SPLINE
SPL {X  -165.650, Y  +580.077, Z    +0.000, E1   -64.018, E3 +192650.768}
SPL {X  -165.650, Y  +590.532, Z    +0.000, E1   -63.993, E3 +192661.334}
SPL {X  -165.650, Y  +600.616, Z    +0.000, E1   -64.059, E3 +192670.908}
SPL {X  -165.650, Y  +609.299, Z    +0.000, E1   -64.001, E3 +192679.933}
SPL {X  -165.650, Y  +618.778, Z    +0.000, E1   -63.957, E3 +192689.790}
SPL {X  -165.650, Y  +634.916, Z    +0.000, E1   -64.117, E3 +192704.838}
SPL {X  -165.650, Y  +648.710, Z    +0.000, E1   -63.999, E3 +192719.249}
SPL {X  -165.650, Y  +658.618, Z    +0.000, E1   -64.006, E3 +192729.066}
SPL {X  -165.650, Y  +670.604, Z    +0.000, E1   -64.021, E3 +192740.979}
SPL {X  -165.270, Y  +686.708, Z    +0.000, E1   -64.001, E3 +192757.322}
SPL {X  -163.641, Y  +701.218, Z    +0.000, E1   -63.638, E3 +192774.466}
SPL {X  -161.003, Y  +714.463, Z    +0.000, E1   -63.428, E3 +192789.138}
SPL {X  -157.854, Y  +725.721, Z    +0.000, E1   -62.989, E3 +192803.387}
SPL {X  -155.984, Y  +731.258, Z    +0.000, E1   -62.241, E3 +192813.532}
SPL {X  -153.281, Y  +738.308, Z    +0.000, E1   -62.233, E3 +192820.720}
SPL {X  -150.070, Y  +745.636, Z    +0.000, E1   -61.982, E3 +192829.467}
SPL {X  -146.912, Y  +752.029, Z    +0.000, E1   -61.155, E3 +192840.569}
SPL {X  -143.078, Y  +758.979, Z    +0.000, E1   -60.553, E3 +192850.549}
SPL {X  -139.815, Y  +764.336, Z    +0.000, E1   -60.025, E3 +192858.400}
SPL {X  -130.672, Y  +777.307, Z    +0.000, E1   -63.098, E3 +192856.691}
SPL {X   -84.123, Y  +818.200, Z    +0.000, E1   -55.499, E3 +192970.205}
ENDSPLINE

SPLINE
SPL {X  -116.242, Y  +793.515, Z    +0.000, E1   -51.439, E3 +193088.077}
SPL {X  -136.975, Y  +768.655, Z    +0.000, E1   -47.464, E3 +193112.533}
SPL {X  -151.617, Y  +742.224, Z    +0.000, E1   -39.442, E3 +193118.920}
SPL {X  -159.277, Y  +721.007, Z    +0.000, E1   -30.118, E3 +193118.098}
SPL {X  -163.701, Y  +700.836, Z    +0.000, E1   -18.960, E3 +193114.812}
SPL {X  -165.229, Y  +687.300, Z    +0.000, E1   -10.302, E3 +193114.768}
SPL {X  -165.635, Y  +677.721, Z    +0.000, E1    -3.517, E3 +193113.899}
SPL {X  -165.650, Y  +672.966, Z    +0.000, E1    +0.394, E3 +193112.802}
SPL {X  -165.650, Y  +668.094, Z    +0.000, E1    +7.098, E3 +193111.985}
SPL {X  -165.650, Y  +662.291, Z    +0.000, E1   +16.729, E3 +193111.910}
SPL {X  -165.650, Y  +656.382, Z    +0.000, E1   +26.732, E3 +193111.468}
SPL {X  -165.650, Y  +648.240, Z    +0.000, E1   +42.276, E3 +193106.902}
SPL {X  -165.650, Y  +638.477, Z    +0.000, E1   +48.488, E3 +193113.403}
SPL {X  -165.650, Y  +615.287, Z    +0.000, E1   +74.123, E3 +193097.934}
SPL {X  -165.650, Y  +589.967, Z    +0.000, E1   +71.395, E3 +193114.277}
SPL {X  -165.650, Y  +573.012, Z    +0.000, E1   +68.475, E3 +193130.490}
SPL {X  -165.650, Y  +459.505, Z    +0.000, E1   +68.780, E3 +193202.214}
ENDSPLINE

SPLINE
SPL {X  -165.650, Y  +483.715, Z    +0.000, E1   +63.891, E3 +193218.508}
ENDSPLINE

SPLINE
SPL {X  -165.650, Y  +474.626, Z    +0.000, E1   +63.707, E3 +193229.037}
SPL {X  -165.650, Y  +465.190, Z    +0.000, E1   +63.660, E3 +193238.892}
SPL {X  -165.650, Y  +456.011, Z    +0.000, E1   +63.585, E3 +193248.786}
SPL {X  -165.650, Y  +444.310, Z    +0.000, E1   +63.666, E3 +193260.064}
SPL {X  -165.650, Y  +429.845, Z    +0.000, E1   +64.481, E3 +193268.297}
SPL {X  -165.552, Y  +372.799, Z    +0.000, E1   +69.633, E3 +193274.161}
SPL {X  -165.443, Y  +370.231, Z    +0.000, E1   +68.724, E3 +193284.091}
SPL {X  -164.908, Y  +362.840, Z    +0.000, E1   +68.443, E3 +193292.436}
SPL {X  -164.361, Y  +357.877, Z    +0.000, E1   +67.700, E3 +193302.891}
SPL {X  -163.803, Y  +353.836, Z    +0.000, E1   +66.282, E3 +193317.912}
SPL {X  -163.046, Y  +349.241, Z    +0.000, E1   +65.245, E3 +193329.838}
SPL {X  -160.229, Y  +336.468, Z    +0.000, E1   +65.236, E3 +193341.821}
SPL {X  -157.078, Y  +325.903, Z    +0.000, E1   +64.692, E3 +193355.266}
SPL {X  -154.296, Y  +318.230, Z    +0.000, E1   +64.302, E3 +193364.823}
SPL {X  -151.091, Y  +310.592, Z    +0.000, E1   +63.929, E3 +193374.274}
SPL {X  -148.836, Y  +305.783, Z    +0.000, E1   +63.120, E3 +193383.406}
SPL {X  -145.492, Y  +299.305, Z    +0.000, E1   +63.037, E3 +193389.898}
SPL {X  -142.120, Y  +293.401, Z    +0.000, E1   +62.602, E3 +193397.578}
SPL {X  -139.854, Y  +289.726, Z    +0.000, E1   +61.679, E3 +193405.483}
SPL {X  -135.997, Y  +283.923, Z    +0.000, E1   +62.034, E3 +193409.132}
SPL {X  -124.991, Y  +269.793, Z    +0.000, E1   +65.852, E3 +193404.122}
SPL {X   -80.641, Y  +233.804, Z    +0.000, E1   +55.283, E3 +193535.236}
ENDSPLINE

SPLINE
SPL {X  -132.197, Y  +278.681, Z    +0.000, E1   +49.692, E3 +193669.109}
SPL {X  -156.075, Y  +322.998, Z    +0.000, E1   +35.140, E3 +193674.190}
SPL {X  -162.799, Y  +347.901, Z    +0.000, E1   +22.644, E3 +193676.696}
SPL {X  -164.930, Y  +363.071, Z    +0.000, E1   +13.041, E3 +193674.436}
SPL {X  -165.571, Y  +373.394, Z    +0.000, E1    +5.725, E3 +193674.777}
SPL {X  -165.650, Y  +380.325, Z    +0.000, E1    +0.301, E3 +193673.073}
SPL {X  -165.650, Y  +383.460, Z    +0.000, E1    -3.790, E3 +193672.300}
SPL {X  -165.650, Y  +389.311, Z    +0.000, E1   -13.234, E3 +193671.785}
SPL {X  -165.650, Y  +395.103, Z    +0.000, E1   -23.932, E3 +193671.078}
SPL {X  -165.650, Y  +401.925, Z    +0.000, E1   -35.470, E3 +193670.345}
SPL {X  -165.650, Y  +410.900, Z    +0.000, E1   -46.977, E3 +193670.962}
SPL {X  -165.650, Y  +423.066, Z    +0.000, E1   -61.140, E3 +193666.693}
SPL {X  -165.650, Y  +461.121, Z    +0.000, E1   -74.504, E3 +193668.042}
SPL {X  -165.650, Y  +487.674, Z    +0.000, E1   -70.215, E3 +193690.853}
SPL {X  -165.650, Y  +585.482, Z    +0.000, E1   -67.026, E3 +193770.016}
ENDSPLINE

SPLINE
SPL {X  -165.650, Y  +571.836, Z    +0.000, E1   -64.066, E3 +193780.036}
ENDSPLINE

SPLINE
SPL {X  -165.650, Y  +580.077, Z    +0.000, E1   -64.018, E3 +193788.699}
SPL {X  -165.650, Y  +590.532, Z    +0.000, E1   -63.993, E3 +193799.265}
SPL {X  -165.650, Y  +604.471, Z    +0.000, E1   -64.071, E3 +193812.773}
SPL {X  -165.650, Y  +618.778, Z    +0.000, E1   -63.957, E3 +193827.721}
SPL {X  -165.650, Y  +627.902, Z    +0.000, E1   -63.871, E3 +193837.447}
SPL {X  -165.650, Y  +640.120, Z    +0.000, E1   -64.248, E3 +193846.788}
SPL {X  -165.650, Y  +648.710, Z    +0.000, E1   -63.999, E3 +193857.180}
SPL {X  -165.650, Y  +660.990, Z    +0.000, E1   -63.976, E3 +193869.705}
SPL {X  -165.633, Y  +677.852, Z    +0.000, E1   -63.999, E3 +193886.478}
SPL {X  -164.651, Y  +693.668, Z    +0.000, E1   -63.860, E3 +193903.310}
SPL {X  -162.406, Y  +708.122, Z    +0.000, E1   -63.726, E3 +193918.604}
SPL {X  -159.930, Y  +718.656, Z    +0.000, E1   -63.142, E3 +193933.215}
SPL {X  -156.651, Y  +729.355, Z    +0.000, E1   -62.675, E3 +193947.051}
SPL {X  -153.281, Y  +738.308, Z    +0.000, E1   -62.233, E3 +193958.651}
SPL {X  -150.070, Y  +745.636, Z    +0.000, E1   -61.982, E3 +193967.398}
SPL {X  -146.912, Y  +752.029, Z    +0.000, E1   -61.155, E3 +193978.500}
SPL {X  -143.078, Y  +758.979, Z    +0.000, E1   -60.553, E3 +193988.480}
SPL {X  -139.815, Y  +764.336, Z    +0.000, E1   -60.025, E3 +193996.332}
SPL {X  -133.503, Y  +773.566, Z    +0.000, E1   -62.412, E3 +193994.458}
SPL {X  -122.896, Y  +786.569, Z    +0.000, E1   -64.831, E3 +193994.618}
SPL {X   -84.123, Y  +818.200, Z    +0.000, E1   -55.499, E3 +194108.136}
ENDSPLINE

SPLINE
SPL {X  -127.502, Y  +781.251, Z    +0.000, E1   -49.821, E3 +194240.269}
SPL {X  -156.175, Y  +730.721, Z    +0.000, E1   -34.737, E3 +194256.548}
SPL {X  -163.040, Y  +704.788, Z    +0.000, E1   -21.201, E3 +194252.248}
SPL {X  -165.038, Y  +689.727, Z    +0.000, E1   -11.987, E3 +194252.895}
SPL {X  -165.635, Y  +677.721, Z    +0.000, E1    -3.517, E3 +194251.830}
SPL {X  -165.650, Y  +672.966, Z    +0.000, E1    +0.394, E3 +194250.733}
SPL {X  -165.650, Y  +668.094, Z    +0.000, E1    +7.098, E3 +194249.916}
SPL {X  -165.650, Y  +661.377, Z    +0.000, E1   +18.170, E3 +194249.856}
SPL {X  -165.650, Y  +654.692, Z    +0.000, E1   +29.740, E3 +194249.104}
SPL {X  -165.650, Y  +648.240, Z    +0.000, E1   +42.276, E3 +194244.833}
SPL {X  -165.650, Y  +638.477, Z    +0.000, E1   +48.488, E3 +194251.334}
SPL {X  -165.650, Y  +615.287, Z    +0.000, E1   +74.123, E3 +194235.865}
SPL {X  -165.650, Y  +589.967, Z    +0.000, E1   +71.395, E3 +194252.208}
SPL {X  -165.650, Y  +573.012, Z    +0.000, E1   +68.475, E3 +194268.421}
SPL {X  -165.650, Y  +459.505, Z    +0.000, E1   +68.780, E3 +194340.145}
ENDSPLINE

SPLINE
SPL {X  -165.650, Y  +483.715, Z    +0.000, E1   +63.891, E3 +194356.439}
ENDSPLINE

SPLINE
SPL {X  -165.650, Y  +474.626, Z    +0.000, E1   +63.707, E3 +194366.968}
SPL {X  -165.650, Y  +465.190, Z    +0.000, E1   +63.660, E3 +194376.823}
SPL {X  -165.650, Y  +456.011, Z    +0.000, E1   +63.585, E3 +194386.717}
SPL {X  -165.650, Y  +441.325, Z    +0.000, E1   +63.847, E3 +194399.687}
SPL {X  -165.552, Y  +372.799, Z    +0.000, E1   +69.633, E3 +194412.092}
SPL {X  -165.443, Y  +370.231, Z    +0.000, E1   +68.724, E3 +194422.022}
SPL {X  -164.776, Y  +361.504, Z    +0.000, E1   +68.225, E3 +194433.497}
SPL {X  -164.241, Y  +356.944, Z    +0.000, E1   +66.930, E3 +194448.020}
SPL {X  -163.312, Y  +350.765, Z    +0.000, E1   +66.182, E3 +194459.196}
SPL {X  -163.046, Y  +349.241, Z    +0.000, E1   +65.245, E3 +194467.769}
SPL {X  -160.229, Y  +336.468, Z    +0.000, E1   +65.236, E3 +194479.752}
SPL {X  -157.078, Y  +325.903, Z    +0.000, E1   +64.692, E3 +194493.197}
SPL {X  -153.279, Y  +315.688, Z    +0.000, E1   +64.219, E3 +194505.770}
SPL {X  -149.447, Y  +307.046, Z    +0.000, E1   +63.460, E3 +194518.355}
SPL {X  -145.492, Y  +299.305, Z    +0.000, E1   +63.037, E3 +194527.829}
SPL {X  -142.120, Y  +293.401, Z    +0.000, E1   +62.602, E3 +194535.509}
SPL {X  -139.854, Y  +289.726, Z    +0.000, E1   +61.679, E3 +194543.414}
SPL {X  -135.997, Y  +283.923, Z    +0.000, E1   +62.034, E3 +194547.064}
SPL {X  -124.991, Y  +269.793, Z    +0.000, E1   +65.852, E3 +194542.053}
SPL {X   -80.641, Y  +233.804, Z    +0.000, E1   +55.283, E3 +194673.167}
ENDSPLINE

SPLINE
SPL {X  -132.197, Y  +278.681, Z    +0.000, E1   +49.692, E3 +194807.040}
SPL {X  -156.075, Y  +322.998, Z    +0.000, E1   +35.140, E3 +194812.121}
SPL {X  -162.799, Y  +347.901, Z    +0.000, E1   +22.644, E3 +194814.627}
SPL {X  -164.930, Y  +363.071, Z    +0.000, E1   +13.041, E3 +194812.367}
SPL {X  -165.629, Y  +375.893, Z    +0.000, E1    +3.908, E3 +194812.224}
SPL {X  -165.650, Y  +380.596, Z    +0.000, E1    -0.052, E3 +194810.906}
SPL {X  -165.650, Y  +383.460, Z    +0.000, E1    -3.790, E3 +194810.231}
SPL {X  -165.650, Y  +389.311, Z    +0.000, E1   -13.234, E3 +194809.716}
SPL {X  -165.650, Y  +395.103, Z    +0.000, E1   -23.932, E3 +194809.009}
SPL {X  -165.650, Y  +401.925, Z    +0.000, E1   -35.470, E3 +194808.276}
SPL {X  -165.650, Y  +410.900, Z    +0.000, E1   -46.977, E3 +194808.893}
SPL {X  -165.650, Y  +420.865, Z    +0.000, E1   -58.704, E3 +194805.785}
SPL {X  -165.650, Y  +450.181, Z    +0.000, E1   -73.218, E3 +194803.732}
SPL {X  -165.650, Y  +487.674, Z    +0.000, E1   -70.215, E3 +194828.784}
SPL {X  -165.650, Y  +590.449, Z    +0.000, E1   -68.990, E3 +194896.729}
ENDSPLINE

SPLINE
SPL {X  -165.650, Y  +577.071, Z    +0.000, E1   -65.152, E3 +194915.052}
ENDSPLINE

SPLINE
SPL {X  -165.650, Y  +580.077, Z    +0.000, E1   -64.018, E3 +194926.630}
SPL {X  -165.650, Y  +590.532, Z    +0.000, E1   -63.993, E3 +194937.196}
SPL {X  -165.650, Y  +600.616, Z    +0.000, E1   -64.059, E3 +194946.770}
SPL {X  -165.650, Y  +609.299, Z    +0.000, E1   -64.001, E3 +194955.795}
SPL {X  -165.650, Y  +618.778, Z    +0.000, E1   -63.957, E3 +194965.652}
SPL {X  -165.650, Y  +634.916, Z    +0.000, E1   -64.117, E3 +194980.700}
SPL {X  -165.650, Y  +648.710, Z    +0.000, E1   -63.999, E3 +194995.111}
SPL {X  -165.650, Y  +658.618, Z    +0.000, E1   -64.006, E3 +195004.928}
SPL {X  -165.650, Y  +670.604, Z    +0.000, E1   -64.021, E3 +195016.841}
SPL {X  -165.270, Y  +686.708, Z    +0.000, E1   -64.001, E3 +195033.184}
SPL {X  -163.641, Y  +701.218, Z    +0.000, E1   -63.638, E3 +195050.328}
SPL {X  -161.003, Y  +714.463, Z    +0.000, E1   -63.428, E3 +195065.000}
SPL {X  -157.854, Y  +725.721, Z    +0.000, E1   -62.989, E3 +195079.249}
SPL {X  -155.984, Y  +731.258, Z    +0.000, E1   -62.241, E3 +195089.395}
SPL {X  -153.281, Y  +738.308, Z    +0.000, E1   -62.233, E3 +195096.582}
SPL {X  -150.070, Y  +745.636, Z    +0.000, E1   -61.982, E3 +195105.329}
SPL {X  -148.438, Y  +749.026, Z    +0.000, E1   -61.150, E3 +195113.335}
SPL {X  -145.760, Y  +754.202, Z    +0.000, E1   -61.108, E3 +195118.752}
SPL {X  -143.078, Y  +758.979, Z    +0.000, E1   -60.553, E3 +195126.411}
SPL {X  -139.815, Y  +764.336, Z    +0.000, E1   -60.025, E3 +195134.263}
SPL {X  -130.672, Y  +777.307, Z    +0.000, E1   -63.098, E3 +195132.553}
SPL {X   -84.123, Y  +818.200, Z    +0.000, E1   -55.499, E3 +195246.067}
ENDSPLINE

SPLINE
SPL {X  -127.502, Y  +781.251, Z    +0.000, E1   -49.821, E3 +195378.200}
SPL {X  -151.617, Y  +742.224, Z    +0.000, E1   -39.442, E3 +195394.782}
SPL {X  -159.277, Y  +721.007, Z    +0.000, E1   -30.118, E3 +195393.960}
SPL {X  -163.701, Y  +700.836, Z    +0.000, E1   -18.960, E3 +195390.674}
SPL {X  -165.229, Y  +687.300, Z    +0.000, E1   -10.302, E3 +195390.630}
SPL {X  -165.592, Y  +679.896, Z    +0.000, E1    -5.071, E3 +195389.910}
SPL {X  -165.650, Y  +674.350, Z    +0.000, E1    -0.828, E3 +195389.284}
SPL {X  -165.650, Y  +672.653, Z    +0.000, E1    +0.827, E3 +195388.477}
SPL {X  -165.650, Y  +668.094, Z    +0.000, E1    +7.098, E3 +195387.847}
SPL {X  -165.650, Y  +662.291, Z    +0.000, E1   +16.729, E3 +195387.772}
SPL {X  -165.650, Y  +656.382, Z    +0.000, E1   +26.732, E3 +195387.330}
SPL {X  -165.650, Y  +648.240, Z    +0.000, E1   +42.276, E3 +195382.765}
SPL {X  -165.650, Y  +638.782, Z    +0.000, E1   +47.719, E3 +195389.974}
SPL {X  -165.650, Y  +622.329, Z    +0.000, E1   +68.753, E3 +195377.514}
SPL {X  -165.650, Y  +589.967, Z    +0.000, E1   +71.395, E3 +195390.139}
SPL {X  -165.650, Y  +573.012, Z    +0.000, E1   +68.475, E3 +195406.352}
SPL {X  -165.650, Y  +459.505, Z    +0.000, E1   +68.780, E3 +195478.076}
ENDSPLINE

SPLINE
SPL {X  -165.650, Y  +483.715, Z    +0.000, E1   +63.891, E3 +195494.370}
ENDSPLINE

SPLINE
SPL {X  -165.650, Y  +474.626, Z    +0.000, E1   +63.707, E3 +195504.899}
SPL {X  -165.650, Y  +465.190, Z    +0.000, E1   +63.660, E3 +195514.754}
SPL {X  -165.650, Y  +456.011, Z    +0.000, E1   +63.585, E3 +195524.648}
SPL {X  -165.650, Y  +444.310, Z    +0.000, E1   +63.666, E3 +195535.926}
SPL {X  -165.650, Y  +429.845, Z    +0.000, E1   +64.481, E3 +195544.159}
SPL {X  -165.552, Y  +372.799, Z    +0.000, E1   +69.633, E3 +195550.023}
SPL {X  -165.188, Y  +366.130, Z    +0.000, E1   +68.611, E3 +195564.426}
SPL {X  -164.361, Y  +357.877, Z    +0.000, E1   +67.700, E3 +195578.753}
SPL {X  -163.803, Y  +353.836, Z    +0.000, E1   +66.282, E3 +195593.774}
SPL {X  -162.254, Y  +345.129, Z    +0.000, E1   +65.301, E3 +195609.224}
SPL {X  -158.875, Y  +331.610, Z    +0.000, E1   +64.945, E3 +195624.283}
SPL {X  -154.872, Y  +319.724, Z    +0.000, E1   +64.496, E3 +195638.197}
SPL {X  -151.091, Y  +310.592, Z    +0.000, E1   +63.929, E3 +195650.136}
SPL {X  -148.836, Y  +305.783, Z    +0.000, E1   +63.120, E3 +195659.268}
SPL {X  -145.492, Y  +299.305, Z    +0.000, E1   +63.037, E3 +195665.760}
SPL {X  -142.120, Y  +293.401, Z    +0.000, E1   +62.602, E3 +195673.440}
SPL {X  -139.854, Y  +289.726, Z    +0.000, E1   +61.679, E3 +195681.345}
SPL {X  -135.997, Y  +283.923, Z    +0.000, E1   +62.034, E3 +195684.995}
SPL {X  -124.991, Y  +269.793, Z    +0.000, E1   +65.852, E3 +195679.984}
SPL {X   -80.641, Y  +233.804, Z    +0.000, E1   +55.283, E3 +195811.098}
ENDSPLINE

SPLINE
SPL {X  -132.197, Y  +278.681, Z    +0.000, E1   +49.692, E3 +195944.971}
SPL {X  -156.075, Y  +322.998, Z    +0.000, E1   +35.140, E3 +195950.052}
SPL {X  -162.799, Y  +347.901, Z    +0.000, E1   +22.644, E3 +195952.558}
SPL {X  -164.930, Y  +363.071, Z    +0.000, E1   +13.041, E3 +195950.298}
SPL {X  -165.629, Y  +375.893, Z    +0.000, E1    +3.908, E3 +195950.155}
SPL {X  -165.650, Y  +380.596, Z    +0.000, E1    -0.052, E3 +195948.837}
SPL {X  -165.650, Y  +383.460, Z    +0.000, E1    -3.790, E3 +195948.162}
SPL {X  -165.650, Y  +389.311, Z    +0.000, E1   -13.234, E3 +195947.647}
SPL {X  -165.650, Y  +395.103, Z    +0.000, E1   -23.932, E3 +195946.940}
SPL {X  -165.650, Y  +401.925, Z    +0.000, E1   -35.470, E3 +195946.207}
SPL {X  -165.650, Y  +410.900, Z    +0.000, E1   -46.977, E3 +195946.824}
SPL {X  -165.650, Y  +423.066, Z    +0.000, E1   -61.140, E3 +195942.555}
SPL {X  -165.650, Y  +461.121, Z    +0.000, E1   -74.504, E3 +195943.904}
SPL {X  -165.650, Y  +487.674, Z    +0.000, E1   -70.215, E3 +195966.715}
SPL {X  -165.650, Y  +585.482, Z    +0.000, E1   -67.026, E3 +196045.878}
ENDSPLINE

SPLINE
SPL {X  -165.650, Y  +571.836, Z    +0.000, E1   -64.066, E3 +196055.898}
ENDSPLINE

SPLINE
SPL {X  -165.650, Y  +580.077, Z    +0.000, E1   -64.018, E3 +196064.561}
SPL {X  -165.650, Y  +590.532, Z    +0.000, E1   -63.993, E3 +196075.127}
SPL {X  -165.650, Y  +604.471, Z    +0.000, E1   -64.071, E3 +196088.635}
SPL {X  -165.650, Y  +618.778, Z    +0.000, E1   -63.957, E3 +196103.583}
SPL {X  -165.650, Y  +627.902, Z    +0.000, E1   -63.871, E3 +196113.309}
SPL {X  -165.650, Y  +640.120, Z    +0.000, E1   -64.248, E3 +196122.650}
SPL {X  -165.650, Y  +648.710, Z    +0.000, E1   -63.999, E3 +196133.042}
SPL {X  -165.650, Y  +660.990, Z    +0.000, E1   -63.976, E3 +196145.567}
SPL {X  -165.633, Y  +677.852, Z    +0.000, E1   -63.999, E3 +196162.340}
SPL {X  -164.651, Y  +693.668, Z    +0.000, E1   -63.860, E3 +196179.173}
SPL {X  -162.406, Y  +708.122, Z    +0.000, E1   -63.726, E3 +196194.467}
SPL {X  -159.930, Y  +718.656, Z    +0.000, E1   -63.142, E3 +196209.077}
SPL {X  -156.651, Y  +729.355, Z    +0.000, E1   -62.675, E3 +196222.913}
SPL {X  -153.281, Y  +738.308, Z    +0.000, E1   -62.233, E3 +196234.513}
SPL {X  -150.070, Y  +745.636, Z    +0.000, E1   -61.982, E3 +196243.260}
SPL {X  -148.438, Y  +749.026, Z    +0.000, E1   -61.150, E3 +196251.266}
SPL {X  -145.760, Y  +754.202, Z    +0.000, E1   -61.108, E3 +196256.683}
SPL {X  -143.078, Y  +758.979, Z    +0.000, E1   -60.553, E3 +196264.342}
SPL {X  -139.815, Y  +764.336, Z    +0.000, E1   -60.025, E3 +196272.194}
SPL {X  -130.672, Y  +777.307, Z    +0.000, E1   -63.098, E3 +196270.484}
SPL {X   -84.123, Y  +818.200, Z    +0.000, E1   -55.499, E3 +196383.998}
ENDSPLINE

SPLINE
SPL {X  -116.242, Y  +793.515, Z    +0.000, E1   -51.439, E3 +196501.871}
SPL {X  -136.975, Y  +768.655, Z    +0.000, E1   -47.464, E3 +196526.326}
SPL {X  -151.617, Y  +742.224, Z    +0.000, E1   -39.442, E3 +196532.713}
SPL {X  -159.277, Y  +721.007, Z    +0.000, E1   -30.118, E3 +196531.891}
SPL {X  -163.701, Y  +700.836, Z    +0.000, E1   -18.960, E3 +196528.605}
SPL {X  -165.229, Y  +687.300, Z    +0.000, E1   -10.302, E3 +196528.561}
SPL {X  -165.635, Y  +677.721, Z    +0.000, E1    -3.517, E3 +196527.692}
SPL {X  -165.650, Y  +673.529, Z    +0.000, E1    -0.069, E3 +196526.820}
SPL {X  -165.650, Y  +671.950, Z    +0.000, E1    +1.795, E3 +196526.189}
SPL {X  -165.650, Y  +668.094, Z    +0.000, E1    +7.098, E3 +196525.778}
SPL {X  -165.650, Y  +661.377, Z    +0.000, E1   +18.170, E3 +196525.718}
SPL {X  -165.650, Y  +654.692, Z    +0.000, E1   +29.740, E3 +196524.966}
SPL {X  -165.650, Y  +648.240, Z    +0.000, E1   +42.276, E3 +196520.696}
SPL {X  -165.650, Y  +638.477, Z    +0.000, E1   +48.488, E3 +196527.196}
SPL {X  -165.650, Y  +615.287, Z    +0.000, E1   +74.123, E3 +196511.727}
SPL {X  -165.650, Y  +589.967, Z    +0.000, E1   +71.395, E3 +196528.070}
SPL {X  -165.650, Y  +573.012, Z    +0.000, E1   +68.475, E3 +196544.283}
SPL {X  -165.650, Y  +459.505, Z    +0.000, E1   +68.780, E3 +196616.007}
ENDSPLINE

SPLINE
SPL {X  -165.650, Y  +483.715, Z    +0.000, E1   +63.891, E3 +196632.301}
ENDSPLINE

SPLINE
SPL {X  -165.650, Y  +474.626, Z    +0.000, E1   +63.707, E3 +196642.830}
SPL {X  -165.650, Y  +465.190, Z    +0.000, E1   +63.660, E3 +196652.685}
SPL {X  -165.650, Y  +456.011, Z    +0.000, E1   +63.585, E3 +196662.579}
SPL {X  -165.650, Y  +441.325, Z    +0.000, E1   +63.847, E3 +196675.549}
SPL {X  -165.552, Y  +372.799, Z    +0.000, E1   +69.633, E3 +196687.954}
SPL {X  -165.443, Y  +370.231, Z    +0.000, E1   +68.724, E3 +196697.884}
SPL {X  -164.908, Y  +362.840, Z    +0.000, E1   +68.443, E3 +196706.229}
SPL {X  -164.361, Y  +357.877, Z    +0.000, E1   +67.700, E3 +196716.684}
SPL {X  -163.803, Y  +353.836, Z    +0.000, E1   +66.282, E3 +196731.705}
SPL {X  -162.254, Y  +345.129, Z    +0.000, E1   +65.301, E3 +196747.155}
SPL {X  -158.875, Y  +331.610, Z    +0.000, E1   +64.945, E3 +196762.214}
SPL {X  -154.872, Y  +319.724, Z    +0.000, E1   +64.496, E3 +196776.128}
SPL {X  -151.091, Y  +310.592, Z    +0.000, E1   +63.929, E3 +196788.067}
SPL {X  -148.836, Y  +305.783, Z    +0.000, E1   +63.120, E3 +196797.199}
SPL {X  -145.492, Y  +299.305, Z    +0.000, E1   +63.037, E3 +196803.691}
SPL {X  -142.120, Y  +293.401, Z    +0.000, E1   +62.602, E3 +196811.371}
SPL {X  -139.854, Y  +289.726, Z    +0.000, E1   +61.679, E3 +196819.276}
SPL {X  -135.997, Y  +283.923, Z    +0.000, E1   +62.034, E3 +196822.926}
SPL {X  -124.991, Y  +269.793, Z    +0.000, E1   +65.852, E3 +196817.915}
SPL {X   -80.641, Y  +233.804, Z    +0.000, E1   +55.283, E3 +196949.029}
ENDSPLINE

SPLINE
SPL {X  -126.633, Y  +271.710, Z    +0.000, E1   +51.055, E3 +197079.495}
SPL {X  -147.744, Y  +303.590, Z    +0.000, E1   +42.717, E3 +197087.987}
SPL {X  -158.730, Y  +331.121, Z    +0.000, E1   +31.334, E3 +197087.895}
SPL {X  -162.799, Y  +347.901, Z    +0.000, E1   +22.644, E3 +197090.489}
SPL {X  -164.930, Y  +363.071, Z    +0.000, E1   +13.041, E3 +197088.229}
SPL {X  -165.629, Y  +375.893, Z    +0.000, E1    +3.908, E3 +197088.086}
SPL {X  -165.650, Y  +380.596, Z    +0.000, E1    -0.052, E3 +197086.768}
SPL {X  -165.650, Y  +383.460, Z    +0.000, E1    -3.790, E3 +197086.093}
SPL {X  -165.650, Y  +387.326, Z    +0.000, E1   -10.041, E3 +197085.964}
SPL {X  -165.650, Y  +392.519, Z    +0.000, E1   -19.014, E3 +197085.118}
SPL {X  -165.650, Y  +401.925, Z    +0.000, E1   -35.470, E3 +197084.138}
SPL {X  -165.650, Y  +410.900, Z    +0.000, E1   -46.977, E3 +197084.756}
SPL {X  -165.650, Y  +420.865, Z    +0.000, E1   -58.704, E3 +197081.647}
SPL {X  -165.650, Y  +450.181, Z    +0.000, E1   -73.218, E3 +197079.594}
SPL {X  -165.650, Y  +487.674, Z    +0.000, E1   -70.215, E3 +197104.646}
SPL {X  -165.650, Y  +590.449, Z    +0.000, E1   -68.990, E3 +197172.591}
ENDSPLINE

SPLINE
SPL {X  -165.650, Y  +577.071, Z    +0.000, E1   -65.152, E3 +197190.914}
ENDSPLINE

SPLINE
SPL {X  -165.650, Y  +580.077, Z    +0.000, E1   -64.018, E3 +197202.492}
SPL {X  -165.650, Y  +590.532, Z    +0.000, E1   -63.993, E3 +197213.058}
SPL {X  -165.650, Y  +604.471, Z    +0.000, E1   -64.071, E3 +197226.566}
SPL {X  -165.650, Y  +618.778, Z    +0.000, E1   -63.957, E3 +197241.514}
SPL {X  -165.650, Y  +627.902, Z    +0.000, E1   -63.871, E3 +197251.240}
SPL {X  -165.650, Y  +640.120, Z    +0.000, E1   -64.248, E3 +197260.581}
SPL {X  -165.650, Y  +648.710, Z    +0.000, E1   -63.999, E3 +197270.973}
SPL {X  -165.650, Y  +658.618, Z    +0.000, E1   -64.006, E3 +197280.790}
SPL {X  -165.650, Y  +670.604, Z    +0.000, E1   -64.021, E3 +197292.703}
SPL {X  -165.270, Y  +686.708, Z    +0.000, E1   -64.001, E3 +197309.046}
SPL {X  -164.361, Y  +696.123, Z    +0.000, E1   -63.520, E3 +197321.757}
SPL {X  -162.406, Y  +708.122, Z    +0.000, E1   -63.726, E3 +197332.398}
SPL {X  -159.930, Y  +718.656, Z    +0.000, E1   -63.142, E3 +197347.008}
SPL {X  -157.142, Y  +727.904, Z    +0.000, E1   -62.905, E3 +197357.697}
SPL {X  -154.742, Y  +734.618, Z    +0.000, E1   -62.412, E3 +197367.596}
SPL {X  -150.939, Y  +743.744, Z    +0.000, E1   -61.955, E3 +197379.537}
SPL {X  -146.912, Y  +752.029, Z    +0.000, E1   -61.155, E3 +197392.293}
SPL {X  -143.078, Y  +758.979, Z    +0.000, E1   -60.553, E3 +197402.273}
SPL {X  -139.815, Y  +764.336, Z    +0.000, E1   -60.025, E3 +197410.125}
SPL {X  -130.672, Y  +777.307, Z    +0.000, E1   -63.098, E3 +197408.415}
SPL {X   -84.123, Y  +818.200, Z    +0.000, E1   -55.499, E3 +197521.929}
ENDSPLINE

SPLINE
SPL {X  -127.502, Y  +781.251, Z    +0.000, E1   -49.821, E3 +197654.062}
SPL {X  -156.175, Y  +730.721, Z    +0.000, E1   -34.737, E3 +197670.341}
SPL {X  -163.701, Y  +700.836, Z    +0.000, E1   -18.960, E3 +197666.536}
SPL {X  -165.229, Y  +687.300, Z    +0.000, E1   -10.302, E3 +197666.492}
SPL {X  -165.592, Y  +679.896, Z    +0.000, E1    -5.071, E3 +197665.772}
SPL {X  -165.650, Y  +673.846, Z    +0.000, E1    -0.441, E3 +197664.852}
SPL {X  -165.650, Y  +670.816, Z    +0.000, E1    +3.131, E3 +197664.143}
SPL {X  -165.650, Y  +666.496, Z    +0.000, E1    +9.886, E3 +197663.217}
SPL {X  -165.650, Y  +662.291, Z    +0.000, E1   +16.729, E3 +197663.634}
SPL {X  -165.650, Y  +656.382, Z    +0.000, E1   +26.732, E3 +197663.192}
SPL {X  -165.650, Y  +648.240, Z    +0.000, E1   +42.276, E3 +197658.627}
SPL {X  -165.650, Y  +638.477, Z    +0.000, E1   +48.488, E3 +197665.127}
SPL {X  -165.650, Y  +615.287, Z    +0.000, E1   +74.123, E3 +197649.658}
SPL {X  -165.650, Y  +589.967, Z    +0.000, E1   +71.395, E3 +197666.001}
SPL {X  -165.650, Y  +573.012, Z    +0.000, E1   +68.475, E3 +197682.214}
SPL {X  -165.650, Y  +459.505, Z    +0.000, E1   +68.780, E3 +197753.938}
ENDSPLINE

SPLINE
SPL {X  -165.650, Y  +483.715, Z    +0.000, E1   +63.891, E3 +197770.232}
ENDSPLINE

SPLINE
SPL {X  -165.650, Y  +474.626, Z    +0.000, E1   +63.707, E3 +197780.761}
SPL {X  -165.650, Y  +465.190, Z    +0.000, E1   +63.660, E3 +197790.616}
SPL {X  -165.650, Y  +456.011, Z    +0.000, E1   +63.585, E3 +197800.510}
SPL {X  -165.650, Y  +441.325, Z    +0.000, E1   +63.847, E3 +197813.480}
SPL {X  -165.552, Y  +372.799, Z    +0.000, E1   +69.633, E3 +197825.885}
SPL {X  -165.443, Y  +370.231, Z    +0.000, E1   +68.724, E3 +197835.815}
SPL {X  -164.776, Y  +361.504, Z    +0.000, E1   +68.225, E3 +197847.290}
SPL {X  -164.241, Y  +356.944, Z    +0.000, E1   +66.930, E3 +197861.813}
SPL {X  -163.312, Y  +350.765, Z    +0.000, E1   +66.182, E3 +197872.989}
SPL {X  -163.046, Y  +349.241, Z    +0.000, E1   +65.245, E3 +197881.562}
SPL {X  -160.229, Y  +336.468, Z    +0.000, E1   +65.236, E3 +197893.545}
SPL {X  -157.078, Y  +325.903, Z    +0.000, E1   +64.692, E3 +197906.991}
SPL {X  -153.279, Y  +315.688, Z    +0.000, E1   +64.219, E3 +197919.563}
SPL {X  -149.447, Y  +307.046, Z    +0.000, E1   +63.460, E3 +197932.148}
SPL {X  -145.492, Y  +299.305, Z    +0.000, E1   +63.037, E3 +197941.622}
SPL {X  -142.120, Y  +293.401, Z    +0.000, E1   +62.602, E3 +197949.302}
SPL {X  -139.854, Y  +289.726, Z    +0.000, E1   +61.679, E3 +197957.207}
SPL {X  -135.997, Y  +283.923, Z    +0.000, E1   +62.034, E3 +197960.857}
SPL {X  -124.991, Y  +269.793, Z    +0.000, E1   +65.852, E3 +197955.846}
SPL {X   -80.641, Y  +233.804, Z    +0.000, E1   +55.283, E3 +198086.960}
ENDSPLINE

SPLINE
SPL {X  -126.633, Y  +271.710, Z    +0.000, E1   +51.055, E3 +198217.426}
SPL {X  -147.744, Y  +303.590, Z    +0.000, E1   +42.717, E3 +198225.918}
SPL {X  -158.730, Y  +331.121, Z    +0.000, E1   +31.334, E3 +198225.826}
SPL {X  -162.799, Y  +347.901, Z    +0.000, E1   +22.644, E3 +198228.420}
SPL {X  -164.930, Y  +363.071, Z    +0.000, E1   +13.041, E3 +198226.160}
SPL {X  -165.629, Y  +375.893, Z    +0.000, E1    +3.908, E3 +198226.017}
SPL {X  -165.650, Y  +381.007, Z    +0.000, E1    -0.398, E3 +198224.557}
SPL {X  -165.650, Y  +385.791, Z    +0.000, E1    -7.347, E3 +198223.918}
SPL {X  -165.650, Y  +390.879, Z    +0.000, E1   -16.263, E3 +198223.205}
SPL {X  -165.650, Y  +395.103, Z    +0.000, E1   -23.932, E3 +198222.803}
SPL {X  -165.650, Y  +401.925, Z    +0.000, E1   -35.470, E3 +198222.069}
SPL {X  -165.650, Y  +410.900, Z    +0.000, E1   -46.977, E3 +198222.687}
SPL {X  -165.650, Y  +423.066, Z    +0.000, E1   -61.140, E3 +198218.417}
SPL {X  -165.650, Y  +461.121, Z    +0.000, E1   -74.504, E3 +198219.766}
SPL {X  -165.650, Y  +487.674, Z    +0.000, E1   -70.215, E3 +198242.577}
SPL {X  -165.650, Y  +585.482, Z    +0.000, E1   -67.026, E3 +198321.740}
ENDSPLINE

SPLINE
SPL {X  -165.650, Y  +571.836, Z    +0.000, E1   -64.066, E3 +198331.760}
ENDSPLINE

SPLINE
SPL {X  -165.650, Y  +580.077, Z    +0.000, E1   -64.018, E3 +198340.423}
SPL {X  -165.650, Y  +590.532, Z    +0.000, E1   -63.993, E3 +198350.989}
SPL {X  -165.650, Y  +600.616, Z    +0.000, E1   -64.059, E3 +198360.563}
SPL {X  -165.650, Y  +609.299, Z    +0.000, E1   -64.001, E3 +198369.588}
SPL {X  -165.650, Y  +618.778, Z    +0.000, E1   -63.957, E3 +198379.445}
SPL {X  -165.650, Y  +627.902, Z    +0.000, E1   -63.871, E3 +198389.171}
SPL {X  -165.650, Y  +640.120, Z    +0.000, E1   -64.248, E3 +198398.512}
SPL {X  -165.650, Y  +648.710, Z    +0.000, E1   -63.999, E3 +198408.904}
SPL {X  -165.650, Y  +658.618, Z    +0.000, E1   -64.006, E3 +198418.721}
SPL {X  -165.650, Y  +670.604, Z    +0.000, E1   -64.021, E3 +198430.635}
SPL {X  -165.553, Y  +681.156, Z    +0.000, E1   -63.834, E3 +198442.509}
SPL {X  -164.651, Y  +693.668, Z    +0.000, E1   -63.860, E3 +198455.035}
SPL {X  -163.017, Y  +704.915, Z    +0.000, E1   -63.665, E3 +198467.477}
SPL {X  -161.003, Y  +714.463, Z    +0.000, E1   -63.428, E3 +198478.793}
SPL {X  -157.854, Y  +725.721, Z    +0.000, E1   -62.989, E3 +198493.042}
SPL {X  -155.984, Y  +731.258, Z    +0.000, E1   -62.241, E3 +198503.188}
SPL {X  -153.281, Y  +738.308, Z    +0.000, E1   -62.233, E3 +198510.375}
SPL {X  -150.070, Y  +745.636, Z    +0.000, E1   -61.982, E3 +198519.122}
SPL {X  -146.912, Y  +752.029, Z    +0.000, E1   -61.155, E3 +198530.224}
SPL {X  -143.078, Y  +758.979, Z    +0.000, E1   -60.553, E3 +198540.204}
SPL {X  -139.815, Y  +764.336, Z    +0.000, E1   -60.025, E3 +198548.056}
SPL {X  -130.672, Y  +777.307, Z    +0.000, E1   -63.098, E3 +198546.346}
SPL {X   -84.123, Y  +818.200, Z    +0.000, E1   -55.499, E3 +198659.860}
ENDSPLINE

SPLINE
SPL {X  -127.502, Y  +781.251, Z    +0.000, E1   -49.821, E3 +198791.993}
SPL {X  -151.617, Y  +742.224, Z    +0.000, E1   -39.442, E3 +198808.575}
SPL {X  -159.277, Y  +721.007, Z    +0.000, E1   -30.118, E3 +198807.753}
SPL {X  -163.701, Y  +700.836, Z    +0.000, E1   -18.960, E3 +198804.467}
SPL {X  -165.229, Y  +687.300, Z    +0.000, E1   -10.302, E3 +198804.423}
SPL {X  -165.592, Y  +679.896, Z    +0.000, E1    -5.071, E3 +198803.704}
SPL {X  -165.650, Y  +673.846, Z    +0.000, E1    -0.441, E3 +198802.783}
SPL {X  -165.650, Y  +670.816, Z    +0.000, E1    +3.131, E3 +198802.074}
SPL {X  -165.650, Y  +666.496, Z    +0.000, E1    +9.886, E3 +198801.148}
SPL {X  -165.650, Y  +661.377, Z    +0.000, E1   +18.170, E3 +198801.580}
SPL {X  -165.650, Y  +654.692, Z    +0.000, E1   +29.740, E3 +198800.828}
SPL {X  -165.650, Y  +648.240, Z    +0.000, E1   +42.276, E3 +198796.558}
SPL {X  -165.650, Y  +638.477, Z    +0.000, E1   +48.488, E3 +198803.058}
SPL {X  -165.650, Y  +615.287, Z    +0.000, E1   +74.123, E3 +198787.589}
SPL {X  -165.650, Y  +589.967, Z    +0.000, E1   +71.395, E3 +198803.932}
SPL {X  -165.650, Y  +573.012, Z    +0.000, E1   +68.475, E3 +198820.145}
SPL {X  -165.650, Y  +459.505, Z    +0.000, E1   +68.780, E3 +198891.869}
ENDSPLINE

SPLINE
SPL {X  -165.650, Y  +483.715, Z    +0.000, E1   +63.891, E3 +198908.163}
ENDSPLINE

SPLINE
SPL {X  -165.650, Y  +474.626, Z    +0.000, E1   +63.707, E3 +198918.692}
SPL {X  -165.650, Y  +465.190, Z    +0.000, E1   +63.660, E3 +198928.547}
SPL {X  -165.650, Y  +456.011, Z    +0.000, E1   +63.585, E3 +198938.441}
SPL {X  -165.650, Y  +444.310, Z    +0.000, E1   +63.666, E3 +198949.719}
SPL {X  -165.650, Y  +429.845, Z    +0.000, E1   +64.481, E3 +198957.952}
SPL {X  -165.552, Y  +372.799, Z    +0.000, E1   +69.633, E3 +198963.816}
SPL {X  -165.188, Y  +366.130, Z    +0.000, E1   +68.611, E3 +198978.219}
SPL {X  -164.361, Y  +357.877, Z    +0.000, E1   +67.700, E3 +198992.546}
SPL {X  -163.803, Y  +353.836, Z    +0.000, E1   +66.282, E3 +199007.567}
SPL {X  -162.254, Y  +345.129, Z    +0.000, E1   +65.301, E3 +199023.017}
SPL {X  -159.503, Y  +333.793, Z    +0.000, E1   +65.139, E3 +199034.462}
SPL {X  -157.078, Y  +325.903, Z    +0.000, E1   +64.692, E3 +199044.922}
SPL {X  -153.279, Y  +315.688, Z    +0.000, E1   +64.219, E3 +199057.494}
SPL {X  -149.447, Y  +307.046, Z    +0.000, E1   +63.460, E3 +199070.079}
SPL {X  -145.492, Y  +299.305, Z    +0.000, E1   +63.037, E3 +199079.553}
SPL {X  -142.120, Y  +293.401, Z    +0.000, E1   +62.602, E3 +199087.233}
SPL {X  -139.854, Y  +289.726, Z    +0.000, E1   +61.679, E3 +199095.138}
SPL {X  -135.997, Y  +283.923, Z    +0.000, E1   +62.034, E3 +199098.788}
SPL {X  -124.991, Y  +269.793, Z    +0.000, E1   +65.852, E3 +199093.777}
SPL {X   -80.641, Y  +233.804, Z    +0.000, E1   +55.283, E3 +199224.891}
ENDSPLINE

SPLINE
SPL {X  -132.197, Y  +278.681, Z    +0.000, E1   +49.692, E3 +199358.764}
SPL {X  -156.075, Y  +322.998, Z    +0.000, E1   +35.140, E3 +199363.845}
SPL {X  -163.642, Y  +352.786, Z    +0.000, E1   +19.725, E3 +199365.624}
SPL {X  -165.477, Y  +370.931, Z    +0.000, E1    +7.630, E3 +199364.213}
SPL {X  -165.650, Y  +378.219, Z    +0.000, E1    +1.951, E3 +199363.485}
SPL {X  -165.650, Y  +380.596, Z    +0.000, E1    -0.052, E3 +199362.630}
SPL {X  -165.650, Y  +383.460, Z    +0.000, E1    -3.790, E3 +199361.955}
SPL {X  -165.650, Y  +387.326, Z    +0.000, E1   -10.041, E3 +199361.826}
SPL {X  -165.650, Y  +392.519, Z    +0.000, E1   -19.014, E3 +199360.980}
SPL {X  -165.650, Y  +401.925, Z    +0.000, E1   -35.470, E3 +199360.001}
SPL {X  -165.650, Y  +410.900, Z    +0.000, E1   -46.977, E3 +199360.618}
SPL {X  -165.650, Y  +420.865, Z    +0.000, E1   -58.704, E3 +199357.509}
SPL {X  -165.650, Y  +450.181, Z    +0.000, E1   -73.218, E3 +199355.456}
SPL {X  -165.650, Y  +487.674, Z    +0.000, E1   -70.215, E3 +199380.508}
SPL {X  -165.650, Y  +585.482, Z    +0.000, E1   -67.026, E3 +199459.671}
ENDSPLINE

SPLINE
SPL {X  -165.650, Y  +577.780, Z    +0.000, E1   -64.060, E3 +199475.883}
ENDSPLINE

SPLINE
SPL {X  -165.650, Y  +590.532, Z    +0.000, E1   -63.993, E3 +199488.920}
SPL {X  -165.650, Y  +600.616, Z    +0.000, E1   -64.059, E3 +199498.494}
SPL {X  -165.650, Y  +609.299, Z    +0.000, E1   -64.001, E3 +199507.519}
SPL {X  -165.650, Y  +618.778, Z    +0.000, E1   -63.957, E3 +199517.376}
SPL {X  -165.650, Y  +627.902, Z    +0.000, E1   -63.871, E3 +199527.102}
SPL {X  -165.650, Y  +640.120, Z    +0.000, E1   -64.248, E3 +199536.443}
SPL {X  -165.650, Y  +648.710, Z    +0.000, E1   -63.999, E3 +199546.835}
SPL {X  -165.650, Y  +658.618, Z    +0.000, E1   -64.006, E3 +199556.652}
SPL {X  -165.650, Y  +670.604, Z    +0.000, E1   -64.021, E3 +199568.566}
SPL {X  -165.553, Y  +681.156, Z    +0.000, E1   -63.834, E3 +199580.440}
SPL {X  -164.651, Y  +693.668, Z    +0.000, E1   -63.860, E3 +199592.966}
SPL {X  -163.017, Y  +704.915, Z    +0.000, E1   -63.665, E3 +199605.408}
SPL {X  -161.003, Y  +714.463, Z    +0.000, E1   -63.428, E3 +199616.724}
SPL {X  -157.854, Y  +725.721, Z    +0.000, E1   -62.989, E3 +199630.973}
SPL {X  -155.984, Y  +731.258, Z    +0.000, E1   -62.241, E3 +199641.119}
SPL {X  -153.281, Y  +738.308, Z    +0.000, E1   -62.233, E3 +199648.306}
SPL {X  -150.070, Y  +745.636, Z    +0.000, E1   -61.982, E3 +199657.053}
SPL {X  -148.438, Y  +749.026, Z    +0.000, E1   -61.150, E3 +199665.060}
SPL {X  -145.760, Y  +754.202, Z    +0.000, E1   -61.108, E3 +199670.476}
SPL {X  -143.078, Y  +758.979, Z    +0.000, E1   -60.553, E3 +199678.135}
SPL {X  -139.815, Y  +764.336, Z    +0.000, E1   -60.025, E3 +199685.987}
SPL {X  -130.672, Y  +777.307, Z    +0.000, E1   -63.098, E3 +199684.277}
SPL {X   -84.123, Y  +818.200, Z    +0.000, E1   -55.499, E3 +199797.791}
ENDSPLINE

SPLINE
SPL {X  -127.502, Y  +781.251, Z    +0.000, E1   -49.821, E3 +199929.924}
SPL {X  -151.617, Y  +742.224, Z    +0.000, E1   -39.442, E3 +199946.506}
SPL {X  -159.277, Y  +721.007, Z    +0.000, E1   -30.118, E3 +199945.684}
SPL {X  -163.701, Y  +700.836, Z    +0.000, E1   -18.960, E3 +199942.399}
SPL {X  -165.229, Y  +687.300, Z    +0.000, E1   -10.302, E3 +199942.354}
SPL {X  -165.592, Y  +679.896, Z    +0.000, E1    -5.071, E3 +199941.635}
SPL {X  -165.650, Y  +673.846, Z    +0.000, E1    -0.441, E3 +199940.714}
SPL {X  -165.650, Y  +671.950, Z    +0.000, E1    +1.795, E3 +199939.982}
SPL {X  -165.650, Y  +668.094, Z    +0.000, E1    +7.098, E3 +199939.571}
SPL {X  -165.650, Y  +661.377, Z    +0.000, E1   +18.170, E3 +199939.511}
SPL {X  -165.650, Y  +654.692, Z    +0.000, E1   +29.740, E3 +199938.759}
SPL {X  -165.650, Y  +648.240, Z    +0.000, E1   +42.276, E3 +199934.489}
SPL {X  -165.650, Y  +638.477, Z    +0.000, E1   +48.488, E3 +199940.989}
SPL {X  -165.650, Y  +615.287, Z    +0.000, E1   +74.123, E3 +199925.520}
SPL {X  -165.650, Y  +589.967, Z    +0.000, E1   +71.395, E3 +199941.863}
SPL {X  -165.650, Y  +573.012, Z    +0.000, E1   +68.475, E3 +199958.076}
SPL {X  -165.650, Y  +459.505, Z    +0.000, E1   +68.780, E3 +200029.800}
ENDSPLINE

SPLINE
SPL {X  -165.650, Y  +483.715, Z    +0.000, E1   +63.891, E3 +200046.094}
ENDSPLINE

SPLINE
SPL {X  -165.650, Y  +474.626, Z    +0.000, E1   +63.707, E3 +200056.623}
SPL {X  -165.650, Y  +465.190, Z    +0.000, E1   +63.660, E3 +200066.478}
SPL {X  -165.650, Y  +456.011, Z    +0.000, E1   +63.585, E3 +200076.372}
SPL {X  -165.650, Y  +444.310, Z    +0.000, E1   +63.666, E3 +200087.650}
SPL {X  -165.650, Y  +429.845, Z    +0.000, E1   +64.481, E3 +200095.883}
SPL {X  -165.552, Y  +372.799, Z    +0.000, E1   +69.633, E3 +200101.747}
SPL {X  -165.188, Y  +366.130, Z    +0.000, E1   +68.611, E3 +200116.150}
SPL {X  -164.361, Y  +357.877, Z    +0.000, E1   +67.700, E3 +200130.477}
SPL {X  -164.353, Y  +357.815, Z    +0.000, E1   +66.333, E3 +200141.378}
SPL {X  -163.312, Y  +350.765, Z    +0.000, E1   +66.182, E3 +200148.851}
SPL {X  -162.254, Y  +345.129, Z    +0.000, E1   +65.301, E3 +200160.948}
SPL {X  -158.875, Y  +331.610, Z    +0.000, E1   +64.945, E3 +200176.007}
SPL {X  -154.872, Y  +319.724, Z    +0.000, E1   +64.496, E3 +200189.921}
SPL {X  -152.078, Y  +312.833, Z    +0.000, E1   +64.044, E3 +200198.970}
SPL {X  -149.447, Y  +307.046, Z    +0.000, E1   +63.460, E3 +200208.010}
SPL {X  -145.492, Y  +299.305, Z    +0.000, E1   +63.037, E3 +200217.485}
SPL {X  -142.120, Y  +293.401, Z    +0.000, E1   +62.602, E3 +200225.164}
SPL {X  -139.854, Y  +289.726, Z    +0.000, E1   +61.679, E3 +200233.069}
SPL {X  -135.997, Y  +283.923, Z    +0.000, E1   +62.034, E3 +200236.719}
SPL {X  -124.991, Y  +269.793, Z    +0.000, E1   +65.852, E3 +200231.708}
SPL {X   -80.641, Y  +233.804, Z    +0.000, E1   +55.283, E3 +200362.823}
ENDSPLINE

SPLINE
SPL {X  -126.633, Y  +271.710, Z    +0.000, E1   +51.055, E3 +200493.288}
SPL {X  -147.744, Y  +303.590, Z    +0.000, E1   +42.717, E3 +200501.780}
SPL {X  -158.730, Y  +331.121, Z    +0.000, E1   +31.334, E3 +200501.688}
SPL {X  -162.799, Y  +347.901, Z    +0.000, E1   +22.644, E3 +200504.282}
SPL {X  -164.930, Y  +363.071, Z    +0.000, E1   +13.041, E3 +200502.022}
SPL {X  -165.571, Y  +373.394, Z    +0.000, E1    +5.725, E3 +200502.363}
SPL {X  -165.650, Y  +380.325, Z    +0.000, E1    +0.301, E3 +200500.659}
SPL {X  -165.650, Y  +383.460, Z    +0.000, E1    -3.790, E3 +200499.886}
SPL {X  -165.650, Y  +389.311, Z    +0.000, E1   -13.234, E3 +200499.372}
SPL {X  -165.650, Y  +395.103, Z    +0.000, E1   -23.932, E3 +200498.665}
SPL {X  -165.650, Y  +401.925, Z    +0.000, E1   -35.470, E3 +200497.932}
SPL {X  -165.650, Y  +410.900, Z    +0.000, E1   -46.977, E3 +200498.549}
SPL {X  -165.650, Y  +423.066, Z    +0.000, E1   -61.140, E3 +200494.280}
SPL {X  -165.650, Y  +461.121, Z    +0.000, E1   -74.504, E3 +200495.628}
SPL {X  -165.650, Y  +487.674, Z    +0.000, E1   -70.215, E3 +200518.439}
SPL {X  -165.650, Y  +585.482, Z    +0.000, E1   -67.026, E3 +200597.602}
ENDSPLINE

SPLINE
SPL {X  -165.650, Y  +571.836, Z    +0.000, E1   -64.066, E3 +200607.622}
ENDSPLINE

SPLINE
SPL {X  -165.650, Y  +580.077, Z    +0.000, E1   -64.018, E3 +200616.285}
SPL {X  -165.650, Y  +590.532, Z    +0.000, E1   -63.993, E3 +200626.851}
SPL {X  -165.650, Y  +604.471, Z    +0.000, E1   -64.071, E3 +200640.359}
SPL {X  -165.650, Y  +618.778, Z    +0.000, E1   -63.957, E3 +200655.307}
SPL {X  -165.650, Y  +627.902, Z    +0.000, E1   -63.871, E3 +200665.033}
SPL {X  -165.650, Y  +640.120, Z    +0.000, E1   -64.248, E3 +200674.374}
SPL {X  -165.650, Y  +648.710, Z    +0.000, E1   -63.999, E3 +200684.766}
SPL {X  -165.650, Y  +660.990, Z    +0.000, E1   -63.976, E3 +200697.292}
SPL {X  -165.633, Y  +677.852, Z    +0.000, E1   -63.999, E3 +200714.064}
SPL {X  -164.651, Y  +693.668, Z    +0.000, E1   -63.860, E3 +200730.897}
SPL {X  -162.406, Y  +708.122, Z    +0.000, E1   -63.726, E3 +200746.191}
SPL {X  -159.930, Y  +718.656, Z    +0.000, E1   -63.142, E3 +200760.801}
SPL {X  -156.651, Y  +729.355, Z    +0.000, E1   -62.675, E3 +200774.637}
SPL {X  -153.281, Y  +738.308, Z    +0.000, E1   -62.233, E3 +200786.237}
SPL {X  -150.070, Y  +745.636, Z    +0.000, E1   -61.982, E3 +200794.984}
SPL {X  -146.912, Y  +752.029, Z    +0.000, E1   -61.155, E3 +200806.086}
SPL {X  -143.078, Y  +758.979, Z    +0.000, E1   -60.553, E3 +200816.066}
SPL {X  -139.815, Y  +764.336, Z    +0.000, E1   -60.025, E3 +200823.918}
SPL {X  -130.672, Y  +777.307, Z    +0.000, E1   -63.098, E3 +200822.208}
SPL {X   -84.123, Y  +818.200, Z    +0.000, E1   -55.499, E3 +200935.722}
ENDSPLINE

SPLINE
SPL {X  -116.242, Y  +793.515, Z    +0.000, E1   -51.439, E3 +201053.595}
SPL {X  -136.975, Y  +768.655, Z    +0.000, E1   -47.464, E3 +201078.050}
SPL {X  -151.617, Y  +742.224, Z    +0.000, E1   -39.442, E3 +201084.437}
SPL {X  -159.277, Y  +721.007, Z    +0.000, E1   -30.118, E3 +201083.615}
SPL {X  -163.701, Y  +700.836, Z    +0.000, E1   -18.960, E3 +201080.330}
SPL {X  -165.229, Y  +687.300, Z    +0.000, E1   -10.302, E3 +201080.285}
SPL {X  -165.635, Y  +677.721, Z    +0.000, E1    -3.517, E3 +201079.416}
SPL {X  -165.650, Y  +673.529, Z    +0.000, E1    -0.069, E3 +201078.544}
SPL {X  -165.650, Y  +670.816, Z    +0.000, E1    +3.131, E3 +201077.936}
SPL {X  -165.650, Y  +666.496, Z    +0.000, E1    +9.886, E3 +201077.010}
SPL {X  -165.650, Y  +662.291, Z    +0.000, E1   +16.729, E3 +201077.427}
SPL {X  -165.650, Y  +656.382, Z    +0.000, E1   +26.732, E3 +201076.985}
SPL {X  -165.650, Y  +648.240, Z    +0.000, E1   +42.276, E3 +201072.420}
SPL {X  -165.650, Y  +638.477, Z    +0.000, E1   +48.488, E3 +201078.920}
SPL {X  -165.650, Y  +615.287, Z    +0.000, E1   +74.123, E3 +201063.451}
SPL {X  -165.650, Y  +589.967, Z    +0.000, E1   +71.395, E3 +201079.795}
SPL {X  -165.650, Y  +573.012, Z    +0.000, E1   +68.475, E3 +201096.007}
SPL {X  -165.650, Y  +459.505, Z    +0.000, E1   +68.780, E3 +201167.731}
ENDSPLINE

SPLINE
SPL {X  -165.650, Y  +483.715, Z    +0.000, E1   +63.891, E3 +201184.025}
ENDSPLINE

SPLINE
SPL {X  -165.650, Y  +474.626, Z    +0.000, E1   +63.707, E3 +201194.554}
SPL {X  -165.650, Y  +465.190, Z    +0.000, E1   +63.660, E3 +201204.409}
SPL {X  -165.650, Y  +456.011, Z    +0.000, E1   +63.585, E3 +201214.303}
SPL {X  -165.650, Y  +444.310, Z    +0.000, E1   +63.666, E3 +201225.581}
SPL {X  -165.650, Y  +429.845, Z    +0.000, E1   +64.481, E3 +201233.814}
SPL {X  -165.552, Y  +372.799, Z    +0.000, E1   +69.633, E3 +201239.678}
SPL {X  -165.443, Y  +370.231, Z    +0.000, E1   +68.724, E3 +201249.608}
SPL {X  -164.776, Y  +361.504, Z    +0.000, E1   +68.225, E3 +201261.083}
SPL {X  -164.241, Y  +356.944, Z    +0.000, E1   +66.930, E3 +201275.606}
SPL {X  -163.312, Y  +350.765, Z    +0.000, E1   +66.182, E3 +201286.782}
SPL {X  -163.046, Y  +349.241, Z    +0.000, E1   +65.245, E3 +201295.355}
SPL {X  -160.229, Y  +336.468, Z    +0.000, E1   +65.236, E3 +201307.338}
SPL {X  -157.078, Y  +325.903, Z    +0.000, E1   +64.692, E3 +201320.784}
SPL {X  -154.296, Y  +318.230, Z    +0.000, E1   +64.302, E3 +201330.340}
SPL {X  -151.091, Y  +310.592, Z    +0.000, E1   +63.929, E3 +201339.792}
SPL {X  -148.836, Y  +305.783, Z    +0.000, E1   +63.120, E3 +201348.923}
SPL {X  -145.492, Y  +299.305, Z    +0.000, E1   +63.037, E3 +201355.416}
SPL {X  -142.120, Y  +293.401, Z    +0.000, E1   +62.602, E3 +201363.095}
SPL {X  -139.854, Y  +289.726, Z    +0.000, E1   +61.679, E3 +201371.000}
SPL {X  -135.997, Y  +283.923, Z    +0.000, E1   +62.034, E3 +201374.650}
SPL {X  -124.991, Y  +269.793, Z    +0.000, E1   +65.852, E3 +201369.639}
SPL {X   -80.641, Y  +233.804, Z    +0.000, E1   +55.283, E3 +201500.754}
ENDSPLINE

SPLINE
SPL {X  -126.633, Y  +271.710, Z    +0.000, E1   +51.055, E3 +201631.219}
SPL {X  -147.744, Y  +303.590, Z    +0.000, E1   +42.717, E3 +201639.711}
SPL {X  -158.730, Y  +331.121, Z    +0.000, E1   +31.334, E3 +201639.619}
SPL {X  -162.799, Y  +347.901, Z    +0.000, E1   +22.644, E3 +201642.213}
SPL {X  -164.930, Y  +363.071, Z    +0.000, E1   +13.041, E3 +201639.953}
SPL {X  -165.571, Y  +373.394, Z    +0.000, E1    +5.725, E3 +201640.294}
SPL {X  -165.650, Y  +380.761, Z    +0.000, E1    -0.041, E3 +201638.438}
SPL {X  -165.650, Y  +385.791, Z    +0.000, E1    -7.347, E3 +201637.711}
SPL {X  -165.650, Y  +390.879, Z    +0.000, E1   -16.263, E3 +201636.998}
SPL {X  -165.650, Y  +395.103, Z    +0.000, E1   -23.932, E3 +201636.596}
SPL {X  -165.650, Y  +401.925, Z    +0.000, E1   -35.470, E3 +201635.863}
SPL {X  -165.650, Y  +410.900, Z    +0.000, E1   -46.977, E3 +201636.480}
SPL {X  -165.650, Y  +420.865, Z    +0.000, E1   -58.704, E3 +201633.371}
SPL {X  -165.650, Y  +450.181, Z    +0.000, E1   -73.218, E3 +201631.318}
SPL {X  -165.650, Y  +487.674, Z    +0.000, E1   -70.215, E3 +201656.370}
SPL {X  -165.650, Y  +590.449, Z    +0.000, E1   -68.990, E3 +201724.315}
ENDSPLINE

SPLINE
SPL {X  -165.650, Y  +577.071, Z    +0.000, E1   -65.152, E3 +201742.639}
ENDSPLINE

SPLINE
SPL {X  -165.650, Y  +580.077, Z    +0.000, E1   -64.018, E3 +201754.217}
SPL {X  -165.650, Y  +590.532, Z    +0.000, E1   -63.993, E3 +201764.782}
SPL {X  -165.650, Y  +604.471, Z    +0.000, E1   -64.071, E3 +201778.290}
SPL {X  -165.650, Y  +618.778, Z    +0.000, E1   -63.957, E3 +201793.238}
SPL {X  -165.650, Y  +627.902, Z    +0.000, E1   -63.871, E3 +201802.964}
SPL {X  -165.650, Y  +640.120, Z    +0.000, E1   -64.248, E3 +201812.305}
SPL {X  -165.650, Y  +648.710, Z    +0.000, E1   -63.999, E3 +201822.697}
SPL {X  -165.650, Y  +658.618, Z    +0.000, E1   -64.006, E3 +201832.514}
SPL {X  -165.650, Y  +670.604, Z    +0.000, E1   -64.021, E3 +201844.428}
SPL {X  -165.270, Y  +686.708, Z    +0.000, E1   -64.001, E3 +201860.771}
SPL {X  -163.641, Y  +701.218, Z    +0.000, E1   -63.638, E3 +201877.915}
SPL {X  -161.003, Y  +714.463, Z    +0.000, E1   -63.428, E3 +201892.586}
SPL {X  -158.978, Y  +722.038, Z    +0.000, E1   -63.038, E3 +201902.654}
SPL {X  -156.651, Y  +729.355, Z    +0.000, E1   -62.675, E3 +201912.568}
SPL {X  -153.281, Y  +738.308, Z    +0.000, E1   -62.233, E3 +201924.169}
SPL {X  -150.070, Y  +745.636, Z    +0.000, E1   -61.982, E3 +201932.915}
SPL {X  -148.438, Y  +749.026, Z    +0.000, E1   -61.150, E3 +201940.922}
SPL {X  -145.760, Y  +754.202, Z    +0.000, E1   -61.108, E3 +201946.338}
SPL {X  -143.078, Y  +758.979, Z    +0.000, E1   -60.553, E3 +201953.997}
SPL {X  -139.815, Y  +764.336, Z    +0.000, E1   -60.025, E3 +201961.849}
SPL {X  -130.672, Y  +777.307, Z    +0.000, E1   -63.098, E3 +201960.140}
SPL {X   -84.123, Y  +818.200, Z    +0.000, E1   -55.499, E3 +202073.653}
ENDSPLINE

SPLINE
SPL {X  -127.502, Y  +781.251, Z    +0.000, E1   -49.821, E3 +202205.786}
SPL {X  -151.617, Y  +742.224, Z    +0.000, E1   -39.442, E3 +202222.368}
SPL {X  -159.277, Y  +721.007, Z    +0.000, E1   -30.118, E3 +202221.546}
SPL {X  -163.701, Y  +700.836, Z    +0.000, E1   -18.960, E3 +202218.261}
SPL {X  -165.229, Y  +687.300, Z    +0.000, E1   -10.302, E3 +202218.216}
SPL {X  -165.592, Y  +679.896, Z    +0.000, E1    -5.071, E3 +202217.497}
SPL {X  -165.650, Y  +673.846, Z    +0.000, E1    -0.441, E3 +202216.576}
SPL {X  -165.650, Y  +670.816, Z    +0.000, E1    +3.131, E3 +202215.867}
SPL {X  -165.650, Y  +666.496, Z    +0.000, E1    +9.886, E3 +202214.941}
SPL {X  -165.650, Y  +661.377, Z    +0.000, E1   +18.170, E3 +202215.373}
SPL {X  -165.650, Y  +654.692, Z    +0.000, E1   +29.740, E3 +202214.621}
SPL {X  -165.650, Y  +648.240, Z    +0.000, E1   +42.276, E3 +202210.351}
SPL {X  -165.650, Y  +638.477, Z    +0.000, E1   +48.488, E3 +202216.851}
SPL {X  -165.650, Y  +615.287, Z    +0.000, E1   +74.123, E3 +202201.382}
SPL {X  -165.650, Y  +589.967, Z    +0.000, E1   +71.395, E3 +202217.726}
SPL {X  -165.650, Y  +573.012, Z    +0.000, E1   +68.475, E3 +202233.938}
SPL {X  -165.650, Y  +459.505, Z    +0.000, E1   +68.780, E3 +202305.662}
ENDSPLINE

SPLINE
SPL {X  -165.650, Y  +483.715, Z    +0.000, E1   +63.891, E3 +202321.956}
ENDSPLINE

SPLINE
SPL {X  -165.650, Y  +474.626, Z    +0.000, E1   +63.707, E3 +202332.485}
SPL {X  -165.650, Y  +465.190, Z    +0.000, E1   +63.660, E3 +202342.340}
SPL {X  -165.650, Y  +456.011, Z    +0.000, E1   +63.585, E3 +202352.234}
SPL {X  -165.650, Y  +444.310, Z    +0.000, E1   +63.666, E3 +202363.512}
SPL {X  -165.650, Y  +429.845, Z    +0.000, E1   +64.481, E3 +202371.745}
SPL {X  -165.552, Y  +372.799, Z    +0.000, E1   +69.633, E3 +202377.609}
SPL {X  -165.188, Y  +366.130, Z    +0.000, E1   +68.611, E3 +202392.012}
SPL {X  -164.361, Y  +357.877, Z    +0.000, E1   +67.700, E3 +202406.339}
SPL {X  -164.353, Y  +357.815, Z    +0.000, E1   +66.333, E3 +202417.240}
SPL {X  -163.312, Y  +350.765, Z    +0.000, E1   +66.182, E3 +202424.713}
SPL {X  -163.046, Y  +349.241, Z    +0.000, E1   +65.245, E3 +202433.286}
SPL {X  -160.229, Y  +336.468, Z    +0.000, E1   +65.236, E3 +202445.269}
SPL {X  -158.158, Y  +329.247, Z    +0.000, E1   +64.622, E3 +202456.040}
SPL {X  -154.872, Y  +319.724, Z    +0.000, E1   +64.496, E3 +202465.783}
SPL {X  -151.091, Y  +310.592, Z    +0.000, E1   +63.929, E3 +202477.723}
SPL {X  -148.836, Y  +305.783, Z    +0.000, E1   +63.120, E3 +202486.854}
SPL {X  -145.492, Y  +299.305, Z    +0.000, E1   +63.037, E3 +202493.347}
SPL {X  -142.120, Y  +293.401, Z    +0.000, E1   +62.602, E3 +202501.026}
SPL {X  -139.854, Y  +289.726, Z    +0.000, E1   +61.679, E3 +202508.931}
SPL {X  -135.997, Y  +283.923, Z    +0.000, E1   +62.034, E3 +202512.581}
SPL {X  -124.991, Y  +269.793, Z    +0.000, E1   +65.852, E3 +202507.570}
SPL {X   -80.641, Y  +233.804, Z    +0.000, E1   +55.283, E3 +202638.685}
ENDSPLINE

SPLINE
SPL {X  -132.197, Y  +278.681, Z    +0.000, E1   +49.692, E3 +202772.557}
SPL {X  -156.075, Y  +322.998, Z    +0.000, E1   +35.140, E3 +202777.638}
SPL {X  -163.642, Y  +352.786, Z    +0.000, E1   +19.725, E3 +202779.417}
SPL {X  -165.477, Y  +370.931, Z    +0.000, E1    +7.630, E3 +202778.006}
SPL {X  -165.650, Y  +378.219, Z    +0.000, E1    +1.951, E3 +202777.278}
SPL {X  -165.650, Y  +381.007, Z    +0.000, E1    -0.398, E3 +202776.281}
SPL {X  -165.650, Y  +385.791, Z    +0.000, E1    -7.347, E3 +202775.642}
SPL {X  -165.650, Y  +390.879, Z    +0.000, E1   -16.263, E3 +202774.929}
SPL {X  -165.650, Y  +395.103, Z    +0.000, E1   -23.932, E3 +202774.527}
SPL {X  -165.650, Y  +401.925, Z    +0.000, E1   -35.470, E3 +202773.794}
SPL {X  -165.650, Y  +410.900, Z    +0.000, E1   -46.977, E3 +202774.411}
SPL {X  -165.650, Y  +423.066, Z    +0.000, E1   -61.140, E3 +202770.142}
SPL {X  -165.650, Y  +461.121, Z    +0.000, E1   -74.504, E3 +202771.490}
SPL {X  -165.650, Y  +487.674, Z    +0.000, E1   -70.215, E3 +202794.301}
SPL {X  -165.650, Y  +585.482, Z    +0.000, E1   -67.026, E3 +202873.464}
ENDSPLINE

SPLINE
SPL {X  -165.650, Y  +577.780, Z    +0.000, E1   -64.060, E3 +202889.676}
ENDSPLINE

SPLINE
SPL {X  -165.650, Y  +590.532, Z    +0.000, E1   -63.993, E3 +202902.713}
SPL {X  -165.650, Y  +600.616, Z    +0.000, E1   -64.059, E3 +202912.287}
SPL {X  -165.650, Y  +609.299, Z    +0.000, E1   -64.001, E3 +202921.312}
SPL {X  -165.650, Y  +618.778, Z    +0.000, E1   -63.957, E3 +202931.169}
SPL {X  -165.650, Y  +627.902, Z    +0.000, E1   -63.871, E3 +202940.895}
SPL {X  -165.650, Y  +640.120, Z    +0.000, E1   -64.248, E3 +202950.236}
SPL {X  -165.650, Y  +648.710, Z    +0.000, E1   -63.999, E3 +202960.628}
SPL {X  -165.650, Y  +658.618, Z    +0.000, E1   -64.006, E3 +202970.445}
SPL {X  -165.650, Y  +670.604, Z    +0.000, E1   -64.021, E3 +202982.359}
SPL {X  -165.270, Y  +686.708, Z    +0.000, E1   -64.001, E3 +202998.702}
SPL {X  -163.641, Y  +701.218, Z    +0.000, E1   -63.638, E3 +203015.846}
SPL {X  -161.003, Y  +714.463, Z    +0.000, E1   -63.428, E3 +203030.517}
SPL {X  -158.978, Y  +722.038, Z    +0.000, E1   -63.038, E3 +203040.585}
SPL {X  -156.651, Y  +729.355, Z    +0.000, E1   -62.675, E3 +203050.500}
SPL {X  -153.281, Y  +738.308, Z    +0.000, E1   -62.233, E3 +203062.100}
SPL {X  -150.070, Y  +745.636, Z    +0.000, E1   -61.982, E3 +203070.846}
SPL {X  -146.912, Y  +752.029, Z    +0.000, E1   -61.155, E3 +203081.948}
SPL {X  -143.078, Y  +758.979, Z    +0.000, E1   -60.553, E3 +203091.928}
SPL {X  -139.815, Y  +764.336, Z    +0.000, E1   -60.025, E3 +203099.780}
SPL {X  -130.672, Y  +777.307, Z    +0.000, E1   -63.098, E3 +203098.071}
SPL {X   -84.123, Y  +818.200, Z    +0.000, E1   -55.499, E3 +203211.584}
ENDSPLINE

SPLINE
SPL {X  -116.242, Y  +793.515, Z    +0.000, E1   -51.439, E3 +203329.457}
SPL {X  -136.975, Y  +768.655, Z    +0.000, E1   -47.464, E3 +203353.912}
SPL {X  -151.617, Y  +742.224, Z    +0.000, E1   -39.442, E3 +203360.299}
SPL {X  -161.699, Y  +711.462, Z    +0.000, E1   -25.093, E3 +203357.307}
SPL {X  -165.038, Y  +689.727, Z    +0.000, E1   -11.987, E3 +203356.344}
SPL {X  -165.592, Y  +679.896, Z    +0.000, E1    -5.071, E3 +203355.428}
SPL {X  -165.650, Y  +674.350, Z    +0.000, E1    -0.828, E3 +203354.802}
SPL {X  -165.650, Y  +672.653, Z    +0.000, E1    +0.827, E3 +203353.994}
SPL {X  -165.650, Y  +669.589, Z    +0.000, E1    +5.031, E3 +203353.824}
SPL {X  -165.650, Y  +666.496, Z    +0.000, E1    +9.886, E3 +203352.872}
SPL {X  -165.650, Y  +662.291, Z    +0.000, E1   +16.729, E3 +203353.289}
SPL {X  -165.650, Y  +656.382, Z    +0.000, E1   +26.732, E3 +203352.847}
SPL {X  -165.650, Y  +648.240, Z    +0.000, E1   +42.276, E3 +203348.282}
SPL {X  -165.650, Y  +638.477, Z    +0.000, E1   +48.488, E3 +203354.782}
SPL {X  -165.650, Y  +615.287, Z    +0.000, E1   +74.123, E3 +203339.313}
SPL {X  -165.650, Y  +589.967, Z    +0.000, E1   +71.395, E3 +203355.657}
SPL {X  -165.650, Y  +573.012, Z    +0.000, E1   +68.475, E3 +203371.869}
SPL {X  -165.650, Y  +459.505, Z    +0.000, E1   +68.780, E3 +203443.593}
ENDSPLINE

SPLINE
SPL {X  -165.650, Y  +483.715, Z    +0.000, E1   +63.891, E3 +203459.887}
ENDSPLINE

SPLINE
SPL {X  -165.650, Y  +474.626, Z    +0.000, E1   +63.707, E3 +203470.416}
SPL {X  -165.650, Y  +465.190, Z    +0.000, E1   +63.660, E3 +203480.271}
SPL {X  -165.650, Y  +456.011, Z    +0.000, E1   +63.585, E3 +203490.165}
SPL {X  -165.650, Y  +441.325, Z    +0.000, E1   +63.847, E3 +203503.135}
SPL {X  -165.552, Y  +372.799, Z    +0.000, E1   +69.633, E3 +203515.540}
SPL {X  -165.188, Y  +366.130, Z    +0.000, E1   +68.611, E3 +203529.943}
SPL {X  -164.361, Y  +357.877, Z    +0.000, E1   +67.700, E3 +203544.270}
SPL {X  -163.803, Y  +353.836, Z    +0.000, E1   +66.282, E3 +203559.291}
SPL {X  -162.254, Y  +345.129, Z    +0.000, E1   +65.301, E3 +203574.741}
SPL {X  -159.503, Y  +333.793, Z    +0.000, E1   +65.139, E3 +203586.186}
SPL {X  -157.078, Y  +325.903, Z    +0.000, E1   +64.692, E3 +203596.646}
SPL {X  -153.279, Y  +315.688, Z    +0.000, E1   +64.219, E3 +203609.218}
SPL {X  -149.447, Y  +307.046, Z    +0.000, E1   +63.460, E3 +203621.803}
SPL {X  -145.492, Y  +299.305, Z    +0.000, E1   +63.037, E3 +203631.278}
SPL {X  -142.120, Y  +293.401, Z    +0.000, E1   +62.602, E3 +203638.957}
SPL {X  -139.854, Y  +289.726, Z    +0.000, E1   +61.679, E3 +203646.862}
SPL {X  -135.997, Y  +283.923, Z    +0.000, E1   +62.034, E3 +203650.512}
SPL {X  -124.991, Y  +269.793, Z    +0.000, E1   +65.852, E3 +203645.501}
SPL {X   -80.641, Y  +233.804, Z    +0.000, E1   +55.283, E3 +203776.616}
ENDSPLINE

SPLINE
SPL {X  -132.197, Y  +278.681, Z    +0.000, E1   +49.692, E3 +203910.488}
SPL {X  -156.075, Y  +322.998, Z    +0.000, E1   +35.140, E3 +203915.569}
SPL {X  -163.642, Y  +352.786, Z    +0.000, E1   +19.725, E3 +203917.348}
SPL {X  -165.477, Y  +370.931, Z    +0.000, E1    +7.630, E3 +203915.937}
SPL {X  -165.650, Y  +378.219, Z    +0.000, E1    +1.951, E3 +203915.209}
SPL {X  -165.650, Y  +380.596, Z    +0.000, E1    -0.052, E3 +203914.354}
SPL {X  -165.650, Y  +383.460, Z    +0.000, E1    -3.790, E3 +203913.679}
SPL {X  -165.650, Y  +387.326, Z    +0.000, E1   -10.041, E3 +203913.551}
SPL {X  -165.650, Y  +392.519, Z    +0.000, E1   -19.014, E3 +203912.704}
SPL {X  -165.650, Y  +401.925, Z    +0.000, E1   -35.470, E3 +203911.725}
SPL {X  -165.650, Y  +410.900, Z    +0.000, E1   -46.977, E3 +203912.342}
SPL {X  -165.650, Y  +420.865, Z    +0.000, E1   -58.704, E3 +203909.233}
SPL {X  -165.650, Y  +450.181, Z    +0.000, E1   -73.218, E3 +203907.180}
SPL {X  -165.650, Y  +487.674, Z    +0.000, E1   -70.215, E3 +203932.232}
SPL {X  -165.650, Y  +585.482, Z    +0.000, E1   -67.026, E3 +204011.395}
ENDSPLINE

SPLINE
SPL {X  -165.650, Y  +577.780, Z    +0.000, E1   -64.060, E3 +204027.607}
ENDSPLINE

SPLINE
SPL {X  -165.650, Y  +590.532, Z    +0.000, E1   -63.993, E3 +204040.644}
SPL {X  -165.650, Y  +600.616, Z    +0.000, E1   -64.059, E3 +204050.218}
SPL {X  -165.650, Y  +609.299, Z    +0.000, E1   -64.001, E3 +204059.243}
SPL {X  -165.650, Y  +618.778, Z    +0.000, E1   -63.957, E3 +204069.100}
SPL {X  -165.650, Y  +634.916, Z    +0.000, E1   -64.117, E3 +204084.148}
SPL {X  -165.650, Y  +648.710, Z    +0.000, E1   -63.999, E3 +204098.559}
SPL {X  -165.650, Y  +658.618, Z    +0.000, E1   -64.006, E3 +204108.376}
SPL {X  -165.650, Y  +670.604, Z    +0.000, E1   -64.021, E3 +204120.290}
SPL {X  -165.553, Y  +681.156, Z    +0.000, E1   -63.834, E3 +204132.164}
SPL {X  -164.651, Y  +693.668, Z    +0.000, E1   -63.860, E3 +204144.690}
SPL {X  -163.017, Y  +704.915, Z    +0.000, E1   -63.665, E3 +204157.132}
SPL {X  -161.003, Y  +714.463, Z    +0.000, E1   -63.428, E3 +204168.448}
SPL {X  -157.854, Y  +725.721, Z    +0.000, E1   -62.989, E3 +204182.697}
SPL {X  -155.984, Y  +731.258, Z    +0.000, E1   -62.241, E3 +204192.843}
SPL {X  -153.281, Y  +738.308, Z    +0.000, E1   -62.233, E3 +204200.031}
SPL {X  -150.070, Y  +745.636, Z    +0.000, E1   -61.982, E3 +204208.777}
SPL {X  -146.912, Y  +752.029, Z    +0.000, E1   -61.155, E3 +204219.879}
SPL {X  -143.078, Y  +758.979, Z    +0.000, E1   -60.553, E3 +204229.859}
SPL {X  -139.815, Y  +764.336, Z    +0.000, E1   -60.025, E3 +204237.711}
SPL {X  -130.672, Y  +777.307, Z    +0.000, E1   -63.098, E3 +204236.002}
SPL {X   -84.123, Y  +818.200, Z    +0.000, E1   -55.499, E3 +204349.515}
ENDSPLINE

SPLINE
SPL {X  -127.502, Y  +781.251, Z    +0.000, E1   -49.821, E3 +204481.648}
SPL {X  -151.617, Y  +742.224, Z    +0.000, E1   -39.442, E3 +204498.230}
SPL {X  -161.699, Y  +711.462, Z    +0.000, E1   -25.093, E3 +204495.238}
SPL {X  -165.038, Y  +689.727, Z    +0.000, E1   -11.987, E3 +204494.275}
SPL {X  -165.635, Y  +677.721, Z    +0.000, E1    -3.517, E3 +204493.209}
SPL {X  -165.650, Y  +673.529, Z    +0.000, E1    -0.069, E3 +204492.337}
SPL {X  -165.650, Y  +671.950, Z    +0.000, E1    +1.795, E3 +204491.706}
SPL {X  -165.650, Y  +668.094, Z    +0.000, E1    +7.098, E3 +204491.295}
SPL {X  -165.650, Y  +661.377, Z    +0.000, E1   +18.170, E3 +204491.235}
SPL {X  -165.650, Y  +654.692, Z    +0.000, E1   +29.740, E3 +204490.483}
SPL {X  -165.650, Y  +648.240, Z    +0.000, E1   +42.276, E3 +204486.213}
SPL {X  -165.650, Y  +638.477, Z    +0.000, E1   +48.488, E3 +204492.713}
SPL {X  -165.650, Y  +615.287, Z    +0.000, E1   +74.123, E3 +204477.244}
SPL {X  -165.650, Y  +589.967, Z    +0.000, E1   +71.395, E3 +204493.588}
SPL {X  -165.650, Y  +573.012, Z    +0.000, E1   +68.475, E3 +204509.800}
SPL {X  -165.650, Y  +459.505, Z    +0.000, E1   +68.780, E3 +204581.524}
ENDSPLINE

SPLINE
SPL {X  -165.650, Y  +483.715, Z    +0.000, E1   +63.891, E3 +204597.818}
ENDSPLINE

SPLINE
SPL {X  -165.650, Y  +474.626, Z    +0.000, E1   +63.707, E3 +204608.347}
SPL {X  -165.650, Y  +465.190, Z    +0.000, E1   +63.660, E3 +204618.202}
SPL {X  -165.650, Y  +456.011, Z    +0.000, E1   +63.585, E3 +204628.097}
SPL {X  -165.650, Y  +441.325, Z    +0.000, E1   +63.847, E3 +204641.066}
SPL {X  -165.552, Y  +372.799, Z    +0.000, E1   +69.633, E3 +204653.471}
SPL {X  -165.443, Y  +370.231, Z    +0.000, E1   +68.724, E3 +204663.401}
SPL {X  -164.908, Y  +362.840, Z    +0.000, E1   +68.443, E3 +204671.747}
SPL {X  -164.361, Y  +357.877, Z    +0.000, E1   +67.700, E3 +204682.201}
SPL {X  -163.803, Y  +353.836, Z    +0.000, E1   +66.282, E3 +204697.222}
SPL {X  -162.254, Y  +345.129, Z    +0.000, E1   +65.301, E3 +204712.672}
SPL {X  -158.875, Y  +331.610, Z    +0.000, E1   +64.945, E3 +204727.731}
SPL {X  -154.872, Y  +319.724, Z    +0.000, E1   +64.496, E3 +204741.645}
SPL {X  -152.078, Y  +312.833, Z    +0.000, E1   +64.044, E3 +204750.694}
SPL {X  -149.447, Y  +307.046, Z    +0.000, E1   +63.460, E3 +204759.735}
SPL {X  -145.492, Y  +299.305, Z    +0.000, E1   +63.037, E3 +204769.209}
SPL {X  -142.120, Y  +293.401, Z    +0.000, E1   +62.602, E3 +204776.888}
SPL {X  -139.854, Y  +289.726, Z    +0.000, E1   +61.679, E3 +204784.793}
SPL {X  -135.997, Y  +283.923, Z    +0.000, E1   +62.034, E3 +204788.443}
SPL {X  -124.991, Y  +269.793, Z    +0.000, E1   +65.852, E3 +204783.432}
SPL {X   -80.641, Y  +233.804, Z    +0.000, E1   +55.283, E3 +204914.547}
ENDSPLINE

SPLINE
SPL {X  -126.633, Y  +271.710, Z    +0.000, E1   +51.055, E3 +205045.012}
SPL {X  -147.744, Y  +303.590, Z    +0.000, E1   +42.717, E3 +205053.504}
SPL {X  -158.730, Y  +331.121, Z    +0.000, E1   +31.334, E3 +205053.413}
SPL {X  -162.799, Y  +347.901, Z    +0.000, E1   +22.644, E3 +205056.006}
SPL {X  -164.930, Y  +363.071, Z    +0.000, E1   +13.041, E3 +205053.746}
SPL {X  -165.571, Y  +373.394, Z    +0.000, E1    +5.725, E3 +205054.087}
SPL {X  -165.650, Y  +380.761, Z    +0.000, E1    -0.041, E3 +205052.231}
SPL {X  -165.650, Y  +385.791, Z    +0.000, E1    -7.347, E3 +205051.505}
SPL {X  -165.650, Y  +390.879, Z    +0.000, E1   -16.263, E3 +205050.791}
SPL {X  -165.650, Y  +395.103, Z    +0.000, E1   -23.932, E3 +205050.389}
SPL {X  -165.650, Y  +401.925, Z    +0.000, E1   -35.470, E3 +205049.656}
SPL {X  -165.650, Y  +410.900, Z    +0.000, E1   -46.977, E3 +205050.273}
SPL {X  -165.650, Y  +423.066, Z    +0.000, E1   -61.140, E3 +205046.004}
SPL {X  -165.650, Y  +461.121, Z    +0.000, E1   -74.504, E3 +205047.352}
SPL {X  -165.650, Y  +487.674, Z    +0.000, E1   -70.215, E3 +205070.164}
SPL {X  -165.650, Y  +585.482, Z    +0.000, E1   -67.026, E3 +205149.326}
ENDSPLINE

SPLINE
SPL {X  -165.650, Y  +577.780, Z    +0.000, E1   -64.060, E3 +205165.538}
ENDSPLINE

SPLINE
SPL {X  -165.650, Y  +590.532, Z    +0.000, E1   -63.993, E3 +205178.575}
SPL {X  -165.650, Y  +600.616, Z    +0.000, E1   -64.059, E3 +205188.149}
SPL {X  -165.650, Y  +609.299, Z    +0.000, E1   -64.001, E3 +205197.174}
SPL {X  -165.650, Y  +618.778, Z    +0.000, E1   -63.957, E3 +205207.031}
SPL {X  -165.650, Y  +634.916, Z    +0.000, E1   -64.117, E3 +205222.079}
SPL {X  -165.650, Y  +648.710, Z    +0.000, E1   -63.999, E3 +205236.490}
SPL {X  -165.650, Y  +658.618, Z    +0.000, E1   -64.006, E3 +205246.307}
SPL {X  -165.650, Y  +670.604, Z    +0.000, E1   -64.021, E3 +205258.221}
SPL {X  -165.270, Y  +686.708, Z    +0.000, E1   -64.001, E3 +205274.564}
SPL {X  -163.641, Y  +701.218, Z    +0.000, E1   -63.638, E3 +205291.708}
SPL {X  -161.003, Y  +714.463, Z    +0.000, E1   -63.428, E3 +205306.379}
SPL {X  -157.854, Y  +725.721, Z    +0.000, E1   -62.989, E3 +205320.628}
SPL {X  -154.742, Y  +734.618, Z    +0.000, E1   -62.412, E3 +205333.114}
SPL {X  -150.939, Y  +743.744, Z    +0.000, E1   -61.955, E3 +205345.055}
SPL {X  -146.912, Y  +752.029, Z    +0.000, E1   -61.155, E3 +205357.810}
SPL {X  -143.078, Y  +758.979, Z    +0.000, E1   -60.553, E3 +205367.790}
SPL {X  -139.815, Y  +764.336, Z    +0.000, E1   -60.025, E3 +205375.642}
SPL {X  -133.503, Y  +773.566, Z    +0.000, E1   -62.412, E3 +205373.768}
SPL {X  -122.896, Y  +786.569, Z    +0.000, E1   -64.831, E3 +205373.928}
SPL {X   -84.728, Y  +817.841, Z    +0.000, E1   -56.970, E3 +205464.605}
ENDSPLINE

SPLINE
SPL {X   -85.913, Y  +817.129, Z    +0.000, E1   -53.985, E3 +205520.864}
SPL {X  -127.502, Y  +781.251, Z    +0.000, E1   -49.821, E3 +205619.579}
SPL {X  -156.175, Y  +730.721, Z    +0.000, E1   -34.737, E3 +205635.858}
SPL {X  -163.040, Y  +704.788, Z    +0.000, E1   -21.201, E3 +205631.558}
SPL {X  -165.038, Y  +689.727, Z    +0.000, E1   -11.987, E3 +205632.206}
SPL {X  -165.635, Y  +677.721, Z    +0.000, E1    -3.517, E3 +205631.140}
SPL {X  -165.650, Y  +673.529, Z    +0.000, E1    -0.069, E3 +205630.268}
SPL {X  -165.650, Y  +670.816, Z    +0.000, E1    +3.131, E3 +205629.660}
SPL {X  -165.650, Y  +666.496, Z    +0.000, E1    +9.886, E3 +205628.734}
SPL {X  -165.650, Y  +662.291, Z    +0.000, E1   +16.729, E3 +205629.151}
SPL {X  -165.650, Y  +656.382, Z    +0.000, E1   +26.732, E3 +205628.709}
SPL {X  -165.650, Y  +648.240, Z    +0.000, E1   +42.276, E3 +205624.144}
SPL {X  -165.650, Y  +638.477, Z    +0.000, E1   +48.488, E3 +205630.644}
SPL {X  -165.650, Y  +615.287, Z    +0.000, E1   +74.123, E3 +205615.175}
SPL {X  -165.650, Y  +589.967, Z    +0.000, E1   +71.395, E3 +205631.519}
SPL {X  -165.650, Y  +573.012, Z    +0.000, E1   +68.475, E3 +205647.731}
SPL {X  -165.650, Y  +459.505, Z    +0.000, E1   +68.780, E3 +205719.455}
ENDSPLINE

SPLINE
SPL {X  -165.650, Y  +483.715, Z    +0.000, E1   +63.891, E3 +205735.749}
ENDSPLINE

SPLINE
SPL {X  -165.650, Y  +474.626, Z    +0.000, E1   +63.707, E3 +205746.278}
SPL {X  -165.650, Y  +465.190, Z    +0.000, E1   +63.660, E3 +205756.133}
SPL {X  -165.650, Y  +456.011, Z    +0.000, E1   +63.585, E3 +205766.028}
SPL {X  -165.650, Y  +441.325, Z    +0.000, E1   +63.847, E3 +205778.997}
SPL {X  -165.552, Y  +372.799, Z    +0.000, E1   +69.633, E3 +205791.402}
SPL {X  -165.443, Y  +370.231, Z    +0.000, E1   +68.724, E3 +205801.332}
SPL {X  -164.776, Y  +361.504, Z    +0.000, E1   +68.225, E3 +205812.807}
SPL {X  -164.241, Y  +356.944, Z    +0.000, E1   +66.930, E3 +205827.330}
SPL {X  -163.312, Y  +350.765, Z    +0.000, E1   +66.182, E3 +205838.506}
SPL {X  -163.046, Y  +349.241, Z    +0.000, E1   +65.245, E3 +205847.079}
SPL {X  -160.229, Y  +336.468, Z    +0.000, E1   +65.236, E3 +205859.062}
SPL {X  -157.078, Y  +325.903, Z    +0.000, E1   +64.692, E3 +205872.508}
SPL {X  -153.279, Y  +315.688, Z    +0.000, E1   +64.219, E3 +205885.080}
SPL {X  -149.447, Y  +307.046, Z    +0.000, E1   +63.460, E3 +205897.666}
SPL {X  -145.492, Y  +299.305, Z    +0.000, E1   +63.037, E3 +205907.140}
SPL {X  -142.120, Y  +293.401, Z    +0.000, E1   +62.602, E3 +205914.819}
SPL {X  -139.854, Y  +289.726, Z    +0.000, E1   +61.679, E3 +205922.725}
SPL {X  -135.997, Y  +283.923, Z    +0.000, E1   +62.034, E3 +205926.374}
SPL {X  -124.991, Y  +269.793, Z    +0.000, E1   +65.852, E3 +205921.363}
SPL {X   -80.641, Y  +233.804, Z    +0.000, E1   +55.283, E3 +206052.478}
ENDSPLINE

SPLINE
SPL {X  -126.633, Y  +271.710, Z    +0.000, E1   +51.055, E3 +206182.943}
SPL {X  -147.744, Y  +303.590, Z    +0.000, E1   +42.717, E3 +206191.436}
SPL {X  -158.730, Y  +331.121, Z    +0.000, E1   +31.334, E3 +206191.344}
SPL {X  -162.799, Y  +347.901, Z    +0.000, E1   +22.644, E3 +206193.937}
SPL {X  -164.930, Y  +363.071, Z    +0.000, E1   +13.041, E3 +206191.677}
SPL {X  -165.629, Y  +375.893, Z    +0.000, E1    +3.908, E3 +206191.534}
SPL {X  -165.650, Y  +380.596, Z    +0.000, E1    -0.052, E3 +206190.216}
SPL {X  -165.650, Y  +383.460, Z    +0.000, E1    -3.790, E3 +206189.541}
SPL {X  -165.650, Y  +387.326, Z    +0.000, E1   -10.041, E3 +206189.413}
SPL {X  -165.650, Y  +392.519, Z    +0.000, E1   -19.014, E3 +206188.566}
SPL {X  -165.650, Y  +401.925, Z    +0.000, E1   -35.470, E3 +206187.587}
SPL {X  -165.650, Y  +410.900, Z    +0.000, E1   -46.977, E3 +206188.204}
SPL {X  -165.650, Y  +420.865, Z    +0.000, E1   -58.704, E3 +206185.095}
SPL {X  -165.650, Y  +450.181, Z    +0.000, E1   -73.218, E3 +206183.042}
SPL {X  -165.650, Y  +487.674, Z    +0.000, E1   -70.215, E3 +206208.095}
SPL {X  -165.650, Y  +590.449, Z    +0.000, E1   -68.990, E3 +206276.039}
ENDSPLINE

SPLINE
SPL {X  -165.650, Y  +577.071, Z    +0.000, E1   -65.152, E3 +206294.363}
ENDSPLINE

SPLINE
SPL {X  -165.650, Y  +580.077, Z    +0.000, E1   -64.018, E3 +206305.941}
SPL {X  -165.650, Y  +590.532, Z    +0.000, E1   -63.993, E3 +206316.507}
SPL {X  -165.650, Y  +604.471, Z    +0.000, E1   -64.071, E3 +206330.014}
SPL {X  -165.650, Y  +618.778, Z    +0.000, E1   -63.957, E3 +206344.962}
SPL {X  -165.650, Y  +634.916, Z    +0.000, E1   -64.117, E3 +206360.010}
SPL {X  -165.650, Y  +648.710, Z    +0.000, E1   -63.999, E3 +206374.421}
SPL {X  -165.650, Y  +658.618, Z    +0.000, E1   -64.006, E3 +206384.238}
SPL {X  -165.650, Y  +670.604, Z    +0.000, E1   -64.021, E3 +206396.152}
SPL {X  -165.553, Y  +681.156, Z    +0.000, E1   -63.834, E3 +206408.027}
SPL {X  -164.902, Y  +691.221, Z    +0.000, E1   -64.073, E3 +206416.285}
SPL {X  -163.641, Y  +701.218, Z    +0.000, E1   -63.638, E3 +206429.639}
SPL {X  -161.003, Y  +714.463, Z    +0.000, E1   -63.428, E3 +206444.310}
SPL {X  -158.978, Y  +722.038, Z    +0.000, E1   -63.038, E3 +206454.378}
SPL {X  -156.651, Y  +729.355, Z    +0.000, E1   -62.675, E3 +206464.293}
SPL {X  -153.281, Y  +738.308, Z    +0.000, E1   -62.233, E3 +206475.893}
SPL {X  -150.070, Y  +745.636, Z    +0.000, E1   -61.982, E3 +206484.639}
SPL {X  -146.912, Y  +752.029, Z    +0.000, E1   -61.155, E3 +206495.741}
SPL {X  -143.078, Y  +758.979, Z    +0.000, E1   -60.553, E3 +206505.721}
SPL {X  -139.815, Y  +764.336, Z    +0.000, E1   -60.025, E3 +206513.573}
SPL {X  -130.672, Y  +777.307, Z    +0.000, E1   -63.098, E3 +206511.864}
SPL {X   -84.123, Y  +818.200, Z    +0.000, E1   -55.499, E3 +206625.377}
ENDSPLINE

SPLINE
SPL {X  -127.502, Y  +781.251, Z    +0.000, E1   -49.821, E3 +206757.510}
SPL {X  -156.175, Y  +730.721, Z    +0.000, E1   -34.737, E3 +206773.789}
SPL {X  -163.701, Y  +700.836, Z    +0.000, E1   -18.960, E3 +206769.985}
SPL {X  -165.229, Y  +687.300, Z    +0.000, E1   -10.302, E3 +206769.940}
SPL {X  -165.635, Y  +677.721, Z    +0.000, E1    -3.517, E3 +206769.071}
SPL {X  -165.650, Y  +672.966, Z    +0.000, E1    +0.394, E3 +206767.974}
SPL {X  -165.650, Y  +668.094, Z    +0.000, E1    +7.098, E3 +206767.157}
SPL {X  -165.650, Y  +662.291, Z    +0.000, E1   +16.729, E3 +206767.082}
SPL {X  -165.650, Y  +656.382, Z    +0.000, E1   +26.732, E3 +206766.640}
SPL {X  -165.650, Y  +648.240, Z    +0.000, E1   +42.276, E3 +206762.075}
SPL {X  -165.650, Y  +638.477, Z    +0.000, E1   +48.488, E3 +206768.575}
SPL {X  -165.650, Y  +615.287, Z    +0.000, E1   +74.123, E3 +206753.106}
SPL {X  -165.650, Y  +589.967, Z    +0.000, E1   +71.395, E3 +206769.450}
SPL {X  -165.650, Y  +573.012, Z    +0.000, E1   +68.475, E3 +206785.662}
SPL {X  -165.650, Y  +459.505, Z    +0.000, E1   +68.780, E3 +206857.386}
ENDSPLINE

SPLINE
SPL {X  -165.650, Y  +483.715, Z    +0.000, E1   +63.891, E3 +206873.680}
ENDSPLINE

SPLINE
SPL {X  -165.650, Y  +474.626, Z    +0.000, E1   +63.707, E3 +206884.209}
SPL {X  -165.650, Y  +465.190, Z    +0.000, E1   +63.660, E3 +206894.064}
SPL {X  -165.650, Y  +456.011, Z    +0.000, E1   +63.585, E3 +206903.959}
SPL {X  -165.650, Y  +441.325, Z    +0.000, E1   +63.847, E3 +206916.928}
SPL {X  -165.552, Y  +372.799, Z    +0.000, E1   +69.633, E3 +206929.334}
SPL {X  -165.188, Y  +366.130, Z    +0.000, E1   +68.611, E3 +206943.736}
SPL {X  -164.361, Y  +357.877, Z    +0.000, E1   +67.700, E3 +206958.063}
SPL {X  -164.353, Y  +357.815, Z    +0.000, E1   +66.333, E3 +206968.964}
SPL {X  -163.312, Y  +350.765, Z    +0.000, E1   +66.182, E3 +206976.437}
SPL {X  -163.046, Y  +349.241, Z    +0.000, E1   +65.245, E3 +206985.010}
SPL {X  -160.229, Y  +336.468, Z    +0.000, E1   +65.236, E3 +206996.993}
SPL {X  -158.158, Y  +329.247, Z    +0.000, E1   +64.622, E3 +207007.764}
SPL {X  -154.872, Y  +319.724, Z    +0.000, E1   +64.496, E3 +207017.507}
SPL {X  -151.091, Y  +310.592, Z    +0.000, E1   +63.929, E3 +207029.447}
SPL {X  -148.836, Y  +305.783, Z    +0.000, E1   +63.120, E3 +207038.578}
SPL {X  -145.492, Y  +299.305, Z    +0.000, E1   +63.037, E3 +207045.071}
SPL {X  -142.120, Y  +293.401, Z    +0.000, E1   +62.602, E3 +207052.750}
SPL {X  -139.854, Y  +289.726, Z    +0.000, E1   +61.679, E3 +207060.656}
SPL {X  -135.997, Y  +283.923, Z    +0.000, E1   +62.034, E3 +207064.305}
SPL {X  -124.991, Y  +269.793, Z    +0.000, E1   +65.852, E3 +207059.294}
SPL {X   -80.641, Y  +233.804, Z    +0.000, E1   +55.283, E3 +207190.409}
ENDSPLINE

SPLINE
SPL {X  -132.197, Y  +278.681, Z    +0.000, E1   +49.692, E3 +207324.281}
SPL {X  -156.075, Y  +322.998, Z    +0.000, E1   +35.140, E3 +207329.362}
SPL {X  -163.642, Y  +352.786, Z    +0.000, E1   +19.725, E3 +207331.141}
SPL {X  -165.477, Y  +370.931, Z    +0.000, E1    +7.630, E3 +207329.730}
SPL {X  -165.650, Y  +378.219, Z    +0.000, E1    +1.951, E3 +207329.002}
SPL {X  -165.650, Y  +380.596, Z    +0.000, E1    -0.052, E3 +207328.147}
SPL {X  -165.650, Y  +383.460, Z    +0.000, E1    -3.790, E3 +207327.472}
SPL {X  -165.650, Y  +387.326, Z    +0.000, E1   -10.041, E3 +207327.344}
SPL {X  -165.650, Y  +392.519, Z    +0.000, E1   -19.014, E3 +207326.497}
SPL {X  -165.650, Y  +401.925, Z    +0.000, E1   -35.470, E3 +207325.518}
SPL {X  -165.650, Y  +410.900, Z    +0.000, E1   -46.977, E3 +207326.135}
SPL {X  -165.650, Y  +420.865, Z    +0.000, E1   -58.704, E3 +207323.026}
SPL {X  -165.650, Y  +450.181, Z    +0.000, E1   -73.218, E3 +207320.973}
SPL {X  -165.650, Y  +487.674, Z    +0.000, E1   -70.215, E3 +207346.026}
SPL {X  -165.650, Y  +590.449, Z    +0.000, E1   -68.990, E3 +207413.971}
ENDSPLINE

SPLINE
SPL {X  -165.650, Y  +577.071, Z    +0.000, E1   -65.152, E3 +207432.294}
ENDSPLINE

SPLINE
SPL {X  -165.650, Y  +580.077, Z    +0.000, E1   -64.018, E3 +207443.872}
SPL {X  -165.650, Y  +590.532, Z    +0.000, E1   -63.993, E3 +207454.438}
SPL {X  -165.650, Y  +604.471, Z    +0.000, E1   -64.071, E3 +207467.945}
SPL {X  -165.650, Y  +618.778, Z    +0.000, E1   -63.957, E3 +207482.893}
SPL {X  -165.650, Y  +627.902, Z    +0.000, E1   -63.871, E3 +207492.620}
SPL {X  -165.650, Y  +640.120, Z    +0.000, E1   -64.248, E3 +207501.960}
SPL {X  -165.650, Y  +648.710, Z    +0.000, E1   -63.999, E3 +207512.352}
SPL {X  -165.650, Y  +660.990, Z    +0.000, E1   -63.976, E3 +207524.878}
SPL {X  -165.633, Y  +677.852, Z    +0.000, E1   -63.999, E3 +207541.651}
SPL {X  -164.651, Y  +693.668, Z    +0.000, E1   -63.860, E3 +207558.483}
SPL {X  -162.406, Y  +708.122, Z    +0.000, E1   -63.726, E3 +207573.777}
SPL {X  -159.930, Y  +718.656, Z    +0.000, E1   -63.142, E3 +207588.387}
SPL {X  -156.651, Y  +729.355, Z    +0.000, E1   -62.675, E3 +207602.224}
SPL {X  -153.281, Y  +738.308, Z    +0.000, E1   -62.233, E3 +207613.824}
SPL {X  -150.070, Y  +745.636, Z    +0.000, E1   -61.982, E3 +207622.570}
SPL {X  -148.438, Y  +749.026, Z    +0.000, E1   -61.150, E3 +207630.577}
SPL {X  -145.760, Y  +754.202, Z    +0.000, E1   -61.108, E3 +207635.993}
SPL {X  -143.078, Y  +758.979, Z    +0.000, E1   -60.553, E3 +207643.652}
SPL {X  -139.815, Y  +764.336, Z    +0.000, E1   -60.025, E3 +207651.504}
SPL {X  -130.672, Y  +777.307, Z    +0.000, E1   -63.098, E3 +207649.795}
SPL {X   -84.123, Y  +818.200, Z    +0.000, E1   -55.499, E3 +207763.308}
ENDSPLINE

SPLINE
SPL {X  -127.502, Y  +781.251, Z    +0.000, E1   -49.821, E3 +207895.441}
SPL {X  -151.617, Y  +742.224, Z    +0.000, E1   -39.442, E3 +207912.024}
SPL {X  -159.277, Y  +721.007, Z    +0.000, E1   -30.118, E3 +207911.201}
SPL {X  -163.701, Y  +700.836, Z    +0.000, E1   -18.960, E3 +207907.916}
SPL {X  -165.229, Y  +687.300, Z    +0.000, E1   -10.302, E3 +207907.871}
SPL {X  -165.592, Y  +679.896, Z    +0.000, E1    -5.071, E3 +207907.152}
SPL {X  -165.650, Y  +674.350, Z    +0.000, E1    -0.828, E3 +207906.526}
SPL {X  -165.650, Y  +672.653, Z    +0.000, E1    +0.827, E3 +207905.718}
SPL {X  -165.650, Y  +668.094, Z    +0.000, E1    +7.098, E3 +207905.088}
SPL {X  -165.650, Y  +662.291, Z    +0.000, E1   +16.729, E3 +207905.013}
SPL {X  -165.650, Y  +656.382, Z    +0.000, E1   +26.732, E3 +207904.572}
SPL {X  -165.650, Y  +648.240, Z    +0.000, E1   +42.276, E3 +207900.006}
SPL {X  -165.650, Y  +638.782, Z    +0.000, E1   +47.719, E3 +207907.216}
SPL {X  -165.650, Y  +622.329, Z    +0.000, E1   +68.753, E3 +207894.755}
SPL {X  -165.650, Y  +589.967, Z    +0.000, E1   +71.395, E3 +207907.381}
SPL {X  -165.650, Y  +573.012, Z    +0.000, E1   +68.475, E3 +207923.593}
SPL {X  -165.650, Y  +459.505, Z    +0.000, E1   +68.780, E3 +207995.317}
ENDSPLINE

SPLINE
SPL {X  -165.650, Y  +483.715, Z    +0.000, E1   +63.891, E3 +208011.611}
ENDSPLINE

SPLINE
SPL {X  -165.650, Y  +474.626, Z    +0.000, E1   +63.707, E3 +208022.140}
SPL {X  -165.650, Y  +465.190, Z    +0.000, E1   +63.660, E3 +208031.995}
SPL {X  -165.650, Y  +456.011, Z    +0.000, E1   +63.585, E3 +208041.890}
SPL {X  -165.650, Y  +441.325, Z    +0.000, E1   +63.847, E3 +208054.859}
SPL {X  -165.552, Y  +372.799, Z    +0.000, E1   +69.633, E3 +208067.265}
SPL {X  -165.443, Y  +370.231, Z    +0.000, E1   +68.724, E3 +208077.194}
SPL {X  -164.776, Y  +361.504, Z    +0.000, E1   +68.225, E3 +208088.669}
SPL {X  -164.241, Y  +356.944, Z    +0.000, E1   +66.930, E3 +208103.192}
SPL {X  -163.312, Y  +350.765, Z    +0.000, E1   +66.182, E3 +208114.368}
SPL {X  -163.046, Y  +349.241, Z    +0.000, E1   +65.245, E3 +208122.941}
SPL {X  -160.229, Y  +336.468, Z    +0.000, E1   +65.236, E3 +208134.924}
SPL {X  -157.078, Y  +325.903, Z    +0.000, E1   +64.692, E3 +208148.370}
SPL {X  -153.279, Y  +315.688, Z    +0.000, E1   +64.219, E3 +208160.943}
SPL {X  -149.447, Y  +307.046, Z    +0.000, E1   +63.460, E3 +208173.528}
SPL {X  -145.492, Y  +299.305, Z    +0.000, E1   +63.037, E3 +208183.002}
SPL {X  -142.120, Y  +293.401, Z    +0.000, E1   +62.602, E3 +208190.681}
SPL {X  -139.854, Y  +289.726, Z    +0.000, E1   +61.679, E3 +208198.587}
SPL {X  -135.997, Y  +283.923, Z    +0.000, E1   +62.034, E3 +208202.236}
SPL {X  -124.991, Y  +269.793, Z    +0.000, E1   +65.852, E3 +208197.225}
SPL {X   -80.641, Y  +233.804, Z    +0.000, E1   +55.283, E3 +208328.340}
ENDSPLINE

SPLINE
SPL {X  -132.197, Y  +278.681, Z    +0.000, E1   +49.692, E3 +208462.212}
SPL {X  -156.075, Y  +322.998, Z    +0.000, E1   +35.140, E3 +208467.293}
SPL {X  -162.799, Y  +347.901, Z    +0.000, E1   +22.644, E3 +208469.799}
SPL {X  -164.930, Y  +363.071, Z    +0.000, E1   +13.041, E3 +208467.539}
SPL {X  -165.629, Y  +375.893, Z    +0.000, E1    +3.908, E3 +208467.397}
SPL {X  -165.650, Y  +380.596, Z    +0.000, E1    -0.052, E3 +208466.078}
SPL {X  -165.650, Y  +383.460, Z    +0.000, E1    -3.790, E3 +208465.403}
SPL {X  -165.650, Y  +389.311, Z    +0.000, E1   -13.234, E3 +208464.889}
SPL {X  -165.650, Y  +395.103, Z    +0.000, E1   -23.932, E3 +208464.182}
SPL {X  -165.650, Y  +401.925, Z    +0.000, E1   -35.470, E3 +208463.449}
SPL {X  -165.650, Y  +410.900, Z    +0.000, E1   -46.977, E3 +208464.066}
SPL {X  -165.650, Y  +420.865, Z    +0.000, E1   -58.704, E3 +208460.957}
SPL {X  -165.650, Y  +450.181, Z    +0.000, E1   -73.218, E3 +208458.904}
SPL {X  -165.650, Y  +487.674, Z    +0.000, E1   -70.215, E3 +208483.957}
SPL {X  -165.650, Y  +590.449, Z    +0.000, E1   -68.990, E3 +208551.902}
ENDSPLINE

SPLINE
SPL {X  -165.650, Y  +577.071, Z    +0.000, E1   -65.152, E3 +208570.225}
ENDSPLINE

SPLINE
SPL {X  -165.650, Y  +580.077, Z    +0.000, E1   -64.018, E3 +208581.803}
SPL {X  -165.650, Y  +590.532, Z    +0.000, E1   -63.993, E3 +208592.369}
SPL {X  -165.650, Y  +600.616, Z    +0.000, E1   -64.059, E3 +208601.942}
SPL {X  -165.650, Y  +609.299, Z    +0.000, E1   -64.001, E3 +208610.967}
SPL {X  -165.650, Y  +618.778, Z    +0.000, E1   -63.957, E3 +208620.824}
SPL {X  -165.650, Y  +634.916, Z    +0.000, E1   -64.117, E3 +208635.873}
SPL {X  -165.650, Y  +648.710, Z    +0.000, E1   -63.999, E3 +208650.283}
SPL {X  -165.650, Y  +658.618, Z    +0.000, E1   -64.006, E3 +208660.100}
SPL {X  -165.650, Y  +670.604, Z    +0.000, E1   -64.021, E3 +208672.014}
SPL {X  -165.270, Y  +686.708, Z    +0.000, E1   -64.001, E3 +208688.357}
SPL {X  -163.641, Y  +701.218, Z    +0.000, E1   -63.638, E3 +208705.501}
SPL {X  -161.003, Y  +714.463, Z    +0.000, E1   -63.428, E3 +208720.172}
SPL {X  -157.854, Y  +725.721, Z    +0.000, E1   -62.989, E3 +208734.421}
SPL {X  -155.984, Y  +731.258, Z    +0.000, E1   -62.241, E3 +208744.567}
SPL {X  -153.281, Y  +738.308, Z    +0.000, E1   -62.233, E3 +208751.755}
SPL {X  -150.070, Y  +745.636, Z    +0.000, E1   -61.982, E3 +208760.501}
SPL {X  -148.438, Y  +749.026, Z    +0.000, E1   -61.150, E3 +208768.508}
SPL {X  -145.760, Y  +754.202, Z    +0.000, E1   -61.108, E3 +208773.924}
SPL {X  -143.078, Y  +758.979, Z    +0.000, E1   -60.553, E3 +208781.583}
SPL {X  -139.815, Y  +764.336, Z    +0.000, E1   -60.025, E3 +208789.435}
SPL {X  -130.672, Y  +777.307, Z    +0.000, E1   -63.098, E3 +208787.726}
SPL {X   -84.123, Y  +818.200, Z    +0.000, E1   -55.499, E3 +208901.239}
ENDSPLINE

SPLINE
SPL {X  -127.502, Y  +781.251, Z    +0.000, E1   -49.821, E3 +209033.372}
SPL {X  -151.617, Y  +742.224, Z    +0.000, E1   -39.442, E3 +209049.955}
SPL {X  -159.277, Y  +721.007, Z    +0.000, E1   -30.118, E3 +209049.132}
SPL {X  -163.701, Y  +700.836, Z    +0.000, E1   -18.960, E3 +209045.847}
SPL {X  -165.229, Y  +687.300, Z    +0.000, E1   -10.302, E3 +209045.802}
SPL {X  -165.592, Y  +679.896, Z    +0.000, E1    -5.071, E3 +209045.083}
SPL {X  -165.650, Y  +674.350, Z    +0.000, E1    -0.828, E3 +209044.457}
SPL {X  -165.650, Y  +672.653, Z    +0.000, E1    +0.827, E3 +209043.649}
SPL {X  -165.650, Y  +668.094, Z    +0.000, E1    +7.098, E3 +209043.019}
SPL {X  -165.650, Y  +662.291, Z    +0.000, E1   +16.729, E3 +209042.945}
SPL {X  -165.650, Y  +656.382, Z    +0.000, E1   +26.732, E3 +209042.503}
SPL {X  -165.650, Y  +648.240, Z    +0.000, E1   +42.276, E3 +209037.937}
SPL {X  -165.650, Y  +638.782, Z    +0.000, E1   +47.719, E3 +209045.147}
SPL {X  -165.650, Y  +622.329, Z    +0.000, E1   +68.753, E3 +209032.686}
SPL {X  -165.650, Y  +589.967, Z    +0.000, E1   +71.395, E3 +209045.312}
SPL {X  -165.650, Y  +573.012, Z    +0.000, E1   +68.475, E3 +209061.524}
SPL {X  -165.650, Y  +459.505, Z    +0.000, E1   +68.780, E3 +209133.248}
ENDSPLINE

SPLINE
SPL {X  -165.650, Y  +483.715, Z    +0.000, E1   +63.891, E3 +209149.542}
ENDSPLINE

SPLINE
SPL {X  -165.650, Y  +474.626, Z    +0.000, E1   +63.707, E3 +209160.071}
SPL {X  -165.650, Y  +465.190, Z    +0.000, E1   +63.660, E3 +209169.926}
SPL {X  -165.650, Y  +456.011, Z    +0.000, E1   +63.585, E3 +209179.821}
SPL {X  -165.650, Y  +441.325, Z    +0.000, E1   +63.847, E3 +209192.790}
SPL {X  -165.552, Y  +372.799, Z    +0.000, E1   +69.633, E3 +209205.196}
SPL {X  -165.443, Y  +370.231, Z    +0.000, E1   +68.724, E3 +209215.125}
SPL {X  -164.776, Y  +361.504, Z    +0.000, E1   +68.225, E3 +209226.600}
SPL {X  -164.241, Y  +356.944, Z    +0.000, E1   +66.930, E3 +209241.123}
SPL {X  -163.312, Y  +350.765, Z    +0.000, E1   +66.182, E3 +209252.300}
SPL {X  -163.046, Y  +349.241, Z    +0.000, E1   +65.245, E3 +209260.872}
SPL {X  -160.229, Y  +336.468, Z    +0.000, E1   +65.236, E3 +209272.855}
SPL {X  -157.078, Y  +325.903, Z    +0.000, E1   +64.692, E3 +209286.301}
SPL {X  -153.279, Y  +315.688, Z    +0.000, E1   +64.219, E3 +209298.874}
SPL {X  -149.447, Y  +307.046, Z    +0.000, E1   +63.460, E3 +209311.459}
SPL {X  -145.492, Y  +299.305, Z    +0.000, E1   +63.037, E3 +209320.933}
SPL {X  -142.120, Y  +293.401, Z    +0.000, E1   +62.602, E3 +209328.612}
SPL {X  -139.854, Y  +289.726, Z    +0.000, E1   +61.679, E3 +209336.518}
SPL {X  -135.997, Y  +283.923, Z    +0.000, E1   +62.034, E3 +209340.167}
SPL {X  -124.991, Y  +269.793, Z    +0.000, E1   +65.852, E3 +209335.156}
SPL {X   -80.641, Y  +233.804, Z    +0.000, E1   +55.283, E3 +209466.271}
ENDSPLINE

SPLINE
SPL {X  -126.633, Y  +271.710, Z    +0.000, E1   +51.055, E3 +209596.737}
SPL {X  -147.744, Y  +303.590, Z    +0.000, E1   +42.717, E3 +209605.229}
SPL {X  -158.730, Y  +331.121, Z    +0.000, E1   +31.334, E3 +209605.137}
SPL {X  -162.799, Y  +347.901, Z    +0.000, E1   +22.644, E3 +209607.730}
SPL {X  -164.930, Y  +363.071, Z    +0.000, E1   +13.041, E3 +209605.470}
SPL {X  -165.629, Y  +375.893, Z    +0.000, E1    +3.908, E3 +209605.328}
SPL {X  -165.650, Y  +380.596, Z    +0.000, E1    -0.052, E3 +209604.009}
SPL {X  -165.650, Y  +383.460, Z    +0.000, E1    -3.790, E3 +209603.334}
SPL {X  -165.650, Y  +387.326, Z    +0.000, E1   -10.041, E3 +209603.206}
SPL {X  -165.650, Y  +392.519, Z    +0.000, E1   -19.014, E3 +209602.359}
SPL {X  -165.650, Y  +401.925, Z    +0.000, E1   -35.470, E3 +209601.380}
SPL {X  -165.650, Y  +410.900, Z    +0.000, E1   -46.977, E3 +209601.997}
SPL {X  -165.650, Y  +420.865, Z    +0.000, E1   -58.704, E3 +209598.888}
SPL {X  -165.650, Y  +450.181, Z    +0.000, E1   -73.218, E3 +209596.835}
SPL {X  -165.650, Y  +487.674, Z    +0.000, E1   -70.215, E3 +209621.888}
SPL {X  -165.650, Y  +585.482, Z    +0.000, E1   -67.026, E3 +209701.050}
ENDSPLINE

SPLINE
SPL {X  -165.650, Y  +571.836, Z    +0.000, E1   -64.066, E3 +209711.070}
ENDSPLINE

SPLINE
SPL {X  -165.650, Y  +580.077, Z    +0.000, E1   -64.018, E3 +209719.734}
SPL {X  -165.650, Y  +590.532, Z    +0.000, E1   -63.993, E3 +209730.300}
SPL {X  -165.650, Y  +604.471, Z    +0.000, E1   -64.071, E3 +209743.807}
SPL {X  -165.650, Y  +618.778, Z    +0.000, E1   -63.957, E3 +209758.755}
SPL {X  -165.650, Y  +634.916, Z    +0.000, E1   -64.117, E3 +209773.804}
SPL {X  -165.650, Y  +648.710, Z    +0.000, E1   -63.999, E3 +209788.214}
SPL {X  -165.650, Y  +658.618, Z    +0.000, E1   -64.006, E3 +209798.031}
SPL {X  -165.650, Y  +670.604, Z    +0.000, E1   -64.021, E3 +209809.945}
SPL {X  -165.270, Y  +686.708, Z    +0.000, E1   -64.001, E3 +209826.288}
SPL {X  -163.641, Y  +701.218, Z    +0.000, E1   -63.638, E3 +209843.432}
SPL {X  -161.003, Y  +714.463, Z    +0.000, E1   -63.428, E3 +209858.103}
SPL {X  -157.854, Y  +725.721, Z    +0.000, E1   -62.989, E3 +209872.352}
SPL {X  -155.984, Y  +731.258, Z    +0.000, E1   -62.241, E3 +209882.498}
SPL {X  -153.281, Y  +738.308, Z    +0.000, E1   -62.233, E3 +209889.686}
SPL {X  -150.070, Y  +745.636, Z    +0.000, E1   -61.982, E3 +209898.432}
SPL {X  -148.438, Y  +749.026, Z    +0.000, E1   -61.150, E3 +209906.439}
SPL {X  -145.760, Y  +754.202, Z    +0.000, E1   -61.108, E3 +209911.855}
SPL {X  -143.078, Y  +758.979, Z    +0.000, E1   -60.553, E3 +209919.514}
SPL {X  -139.815, Y  +764.336, Z    +0.000, E1   -60.025, E3 +209927.366}
SPL {X  -130.672, Y  +777.307, Z    +0.000, E1   -63.098, E3 +209925.657}
SPL {X   -84.123, Y  +818.200, Z    +0.000, E1   -55.499, E3 +210039.170}
ENDSPLINE

SPLINE
SPL {X  -127.502, Y  +781.251, Z    +0.000, E1   -49.821, E3 +210171.303}
SPL {X  -151.617, Y  +742.224, Z    +0.000, E1   -39.442, E3 +210187.886}
SPL {X  -159.277, Y  +721.007, Z    +0.000, E1   -30.118, E3 +210187.063}
SPL {X  -163.701, Y  +700.836, Z    +0.000, E1   -18.960, E3 +210183.778}
SPL {X  -165.229, Y  +687.300, Z    +0.000, E1   -10.302, E3 +210183.733}
SPL {X  -165.592, Y  +679.896, Z    +0.000, E1    -5.071, E3 +210183.014}
SPL {X  -165.650, Y  +674.350, Z    +0.000, E1    -0.828, E3 +210182.388}
SPL {X  -165.650, Y  +672.653, Z    +0.000, E1    +0.827, E3 +210181.581}
SPL {X  -165.650, Y  +668.094, Z    +0.000, E1    +7.098, E3 +210180.950}
SPL {X  -165.650, Y  +662.291, Z    +0.000, E1   +16.729, E3 +210180.876}
SPL {X  -165.650, Y  +656.382, Z    +0.000, E1   +26.732, E3 +210180.434}
SPL {X  -165.650, Y  +648.240, Z    +0.000, E1   +42.276, E3 +210175.868}
SPL {X  -165.650, Y  +638.782, Z    +0.000, E1   +47.719, E3 +210183.078}
SPL {X  -165.650, Y  +622.329, Z    +0.000, E1   +68.753, E3 +210170.617}
SPL {X  -165.650, Y  +589.967, Z    +0.000, E1   +71.395, E3 +210183.243}
SPL {X  -165.650, Y  +573.012, Z    +0.000, E1   +68.475, E3 +210199.455}
SPL {X  -165.650, Y  +459.505, Z    +0.000, E1   +68.780, E3 +210271.179}
ENDSPLINE

SPLINE
SPL {X  -165.650, Y  +483.715, Z    +0.000, E1   +63.891, E3 +210287.473}
ENDSPLINE

SPLINE
SPL {X  -165.650, Y  +474.626, Z    +0.000, E1   +63.707, E3 +210298.002}
SPL {X  -165.650, Y  +465.190, Z    +0.000, E1   +63.660, E3 +210307.857}
SPL {X  -165.650, Y  +456.011, Z    +0.000, E1   +63.585, E3 +210317.752}
SPL {X  -165.650, Y  +444.310, Z    +0.000, E1   +63.666, E3 +210329.029}
SPL {X  -165.650, Y  +429.845, Z    +0.000, E1   +64.481, E3 +210337.262}
SPL {X  -165.552, Y  +372.799, Z    +0.000, E1   +69.633, E3 +210343.127}
SPL {X  -165.188, Y  +366.130, Z    +0.000, E1   +68.611, E3 +210357.529}
SPL {X  -164.361, Y  +357.877, Z    +0.000, E1   +67.700, E3 +210371.856}
SPL {X  -163.803, Y  +353.836, Z    +0.000, E1   +66.282, E3 +210386.877}
ENDSPLINE

SPLINE
SPL {X  -165.650, Y  +379.091, Z    +0.000, E1   +60.866, E3 +210400.592}
ENDSPLINE

SPLINE
SPL {X  -165.125, Y  +365.326, Z    +0.000, E1   +61.696, E3 +210410.198}
SPL {X  -164.823, Y  +361.969, Z    +0.000, E1   +60.899, E3 +210419.432}
SPL {X  -163.414, Y  +351.372, Z    +0.000, E1   +61.284, E3 +210428.695}
SPL {X  -162.189, Y  +344.818, Z    +0.000, E1   +60.900, E3 +210438.548}
SPL {X  -160.769, Y  +338.584, Z    +0.000, E1   +60.413, E3 +210448.724}
SPL {X  -157.780, Y  +328.049, Z    +0.000, E1   +60.445, E3 +210460.391}
SPL {X  -155.286, Y  +320.826, Z    +0.000, E1   +59.686, E3 +210472.946}
SPL {X  -152.445, Y  +313.689, Z    +0.000, E1   +59.490, E3 +210482.012}
SPL {X  -150.678, Y  +309.680, Z    +0.000, E1   +58.971, E3 +210489.324}
SPL {X  -148.010, Y  +304.117, Z    +0.000, E1   +58.696, E3 +210497.071}
SPL {X  -144.822, Y  +298.086, Z    +0.000, E1   +58.093, E3 +210506.853}
SPL {X  -142.530, Y  +294.089, Z    +0.000, E1   +57.567, E3 +210513.737}
SPL {X  -136.453, Y  +284.583, Z    +0.000, E1   +60.257, E3 +210511.548}
SPL {X  -128.205, Y  +273.602, Z    +0.000, E1   +62.388, E3 +210512.251}
SPL {X   -93.591, Y  +241.823, Z    +0.000, E1   +55.455, E3 +210604.381}
ENDSPLINE

SPLINE
SPL {X  -110.554, Y  +255.140, Z    +0.000, E1   +52.082, E3 +210731.337}
SPL {X  -137.038, Y  +285.439, Z    +0.000, E1   +46.261, E3 +210751.076}
SPL {X  -149.954, Y  +308.117, Z    +0.000, E1   +39.560, E3 +210757.424}
SPL {X  -160.070, Y  +335.868, Z    +0.000, E1   +27.320, E3 +210751.823}
SPL {X  -163.969, Y  +354.959, Z    +0.000, E1   +17.178, E3 +210752.337}
SPL {X  -165.261, Y  +367.153, Z    +0.000, E1    +9.611, E3 +210751.489}
SPL {X  -165.600, Y  +374.440, Z    +0.000, E1    +4.699, E3 +210750.750}
SPL {X  -165.650, Y  +379.657, Z    +0.000, E1    +0.819, E3 +210750.279}
SPL {X  -165.650, Y  +381.885, Z    +0.000, E1    -1.282, E3 +210749.523}
SPL {X  -165.650, Y  +386.855, Z    +0.000, E1    -7.700, E3 +210748.942}
SPL {X  -165.650, Y  +393.198, Z    +0.000, E1   -17.733, E3 +210747.918}
SPL {X  -165.650, Y  +399.991, Z    +0.000, E1   -27.922, E3 +210748.814}
SPL {X  -165.650, Y  +411.457, Z    +0.000, E1   -45.557, E3 +210744.561}
SPL {X  -165.650, Y  +427.627, Z    +0.000, E1   -58.747, E3 +210745.196}
SPL {X  -165.650, Y  +479.770, Z    +0.000, E1   -67.621, E3 +210765.810}
SPL {X  -165.650, Y  +594.725, Z    +0.000, E1   -69.155, E3 +210833.271}
ENDSPLINE

SPLINE
SPL {X  -165.650, Y  +565.175, Z    +0.000, E1   -62.653, E3 +210856.762}
ENDSPLINE

SPLINE
SPL {X  -165.650, Y  +576.067, Z    +0.000, E1   -62.373, E3 +210870.163}
SPL {X  -165.650, Y  +586.101, Z    +0.000, E1   -62.398, E3 +210880.745}
SPL {X  -165.650, Y  +596.110, Z    +0.000, E1   -62.302, E3 +210892.186}
SPL {X  -165.650, Y  +607.052, Z    +0.000, E1   -62.387, E3 +210903.253}
SPL {X  -165.650, Y  +618.920, Z    +0.000, E1   -62.340, E3 +210916.444}
SPL {X  -165.650, Y  +631.247, Z    +0.000, E1   -62.270, E3 +210930.060}
SPL {X  -165.650, Y  +645.288, Z    +0.000, E1   -62.475, E3 +210943.740}
SPL {X  -165.650, Y  +657.265, Z    +0.000, E1   -62.410, E3 +210956.859}
SPL {X  -165.650, Y  +665.926, Z    +0.000, E1   -62.171, E3 +210967.872}
SPL {X  -165.600, Y  +679.566, Z    +0.000, E1   -62.408, E3 +210980.910}
SPL {X  -165.066, Y  +689.394, Z    +0.000, E1   -62.143, E3 +210993.239}
SPL {X  -164.056, Y  +698.425, Z    +0.000, E1   -62.113, E3 +211003.159}
SPL {X  -162.891, Y  +705.608, Z    +0.000, E1   -61.899, E3 +211012.331}
SPL {X  -161.308, Y  +713.180, Z    +0.000, E1   -61.813, E3 +211021.024}
SPL {X  -159.339, Y  +720.787, Z    +0.000, E1   -61.452, E3 +211031.720}
SPL {X  -156.103, Y  +730.922, Z    +0.000, E1   -60.875, E3 +211046.266}
SPL {X  -152.882, Y  +739.274, Z    +0.000, E1   -60.485, E3 +211057.448}
SPL {X  -150.387, Y  +744.953, Z    +0.000, E1   -60.023, E3 +211066.123}
SPL {X  -146.839, Y  +752.170, Z    +0.000, E1   -59.458, E3 +211077.082}
SPL {X  -142.415, Y  +760.104, Z    +0.000, E1   -58.730, E3 +211089.140}
SPL {X  -134.606, Y  +772.046, Z    +0.000, E1   -61.105, E3 +211090.470}
SPL {X  -127.075, Y  +781.763, Z    +0.000, E1   -62.555, E3 +211092.784}
SPL {X   -89.692, Y  +814.767, Z    +0.000, E1   -54.641, E3 +211205.258}
ENDSPLINE

SPLINE
SPL {X  -133.336, Y  +773.792, Z    +0.000, E1   -47.991, E3 +211333.725}
SPL {X  -153.017, Y  +738.949, Z    +0.000, E1   -37.928, E3 +211347.129}
SPL {X  -160.146, Y  +717.846, Z    +0.000, E1   -27.412, E3 +211334.675}
SPL {X  -163.639, Y  +701.236, Z    +0.000, E1   -18.901, E3 +211340.817}
SPL {X  -165.380, Y  +684.951, Z    +0.000, E1    -8.606, E3 +211339.074}
SPL {X  -165.650, Y  +675.640, Z    +0.000, E1    -1.874, E3 +211338.610}
SPL {X  -165.650, Y  +673.425, Z    +0.000, E1    +0.051, E3 +211337.616}
SPL {X  -165.650, Y  +672.004, Z    +0.000, E1    +1.620, E3 +211337.094}
SPL {X  -165.650, Y  +669.258, Z    +0.000, E1    +5.269, E3 +211336.713}
SPL {X  -165.650, Y  +665.011, Z    +0.000, E1   +11.627, E3 +211336.600}
SPL {X  -165.650, Y  +659.446, Z    +0.000, E1   +21.123, E3 +211335.464}
SPL {X  -165.650, Y  +651.038, Z    +0.000, E1   +34.281, E3 +211335.090}
SPL {X  -165.650, Y  +635.255, Z    +0.000, E1   +53.641, E3 +211333.278}
SPL {X  -165.650, Y  +581.672, Z    +0.000, E1   +69.744, E3 +211345.685}
SPL {X  -165.650, Y  +455.882, Z    +0.000, E1   +70.075, E3 +211417.950}
ENDSPLINE

SPLINE
SPL {X  -165.650, Y  +480.501, Z    +0.000, E1   +64.561, E3 +211439.919}
ENDSPLINE

SPLINE
SPL {X  -165.650, Y  +477.868, Z    +0.000, E1   +63.324, E3 +211451.846}
SPL {X  -165.650, Y  +463.578, Z    +0.000, E1   +63.625, E3 +211464.200}
SPL {X  -165.650, Y  +453.769, Z    +0.000, E1   +63.450, E3 +211475.459}
SPL {X  -165.650, Y  +444.234, Z    +0.000, E1   +63.262, E3 +211486.632}
SPL {X  -165.650, Y  +432.479, Z    +0.000, E1   +63.557, E3 +211496.452}
SPL {X  -165.650, Y  +422.068, Z    +0.000, E1   +63.630, E3 +211506.547}
SPL {X  -165.650, Y  +409.231, Z    +0.000, E1   +63.364, E3 +211521.796}
SPL {X  -165.650, Y  +395.008, Z    +0.000, E1   +63.445, E3 +211535.559}
ENDSPLINE

SPLINE
SPL {X  -165.650, Y  +410.094, Z    +0.000, E1   +60.049, E3 +211543.008}
ENDSPLINE

SPLINE
SPL {X  -165.650, Y  +398.700, Z    +0.000, E1   +60.415, E3 +211553.906}
SPL {X  -165.650, Y  +380.643, Z    +0.000, E1   +61.187, E3 +211569.268}
SPL {X  -165.125, Y  +365.326, Z    +0.000, E1   +61.696, E3 +211582.611}
SPL {X  -164.823, Y  +361.969, Z    +0.000, E1   +60.899, E3 +211591.846}
SPL {X  -163.414, Y  +351.372, Z    +0.000, E1   +61.284, E3 +211601.109}
SPL {X  -162.189, Y  +344.818, Z    +0.000, E1   +60.900, E3 +211610.962}
SPL {X  -160.769, Y  +338.584, Z    +0.000, E1   +60.413, E3 +211621.138}
SPL {X  -157.780, Y  +328.049, Z    +0.000, E1   +60.445, E3 +211632.805}
SPL {X  -155.286, Y  +320.826, Z    +0.000, E1   +59.686, E3 +211645.360}
SPL {X  -152.445, Y  +313.689, Z    +0.000, E1   +59.490, E3 +211654.426}
SPL {X  -149.851, Y  +307.898, Z    +0.000, E1   +58.978, E3 +211663.748}
SPL {X  -146.926, Y  +301.997, Z    +0.000, E1   +58.334, E3 +211673.709}
SPL {X  -143.281, Y  +295.370, Z    +0.000, E1   +57.860, E3 +211683.478}
SPL {X  -134.010, Y  +281.128, Z    +0.000, E1   +60.923, E3 +211684.256}
SPL {X   -93.591, Y  +241.823, Z    +0.000, E1   +55.455, E3 +211776.794}
ENDSPLINE

SPLINE
SPL {X  -110.554, Y  +255.140, Z    +0.000, E1   +52.082, E3 +211903.750}
SPL {X  -137.038, Y  +285.439, Z    +0.000, E1   +46.261, E3 +211923.490}
SPL {X  -149.954, Y  +308.117, Z    +0.000, E1   +39.560, E3 +211929.838}
SPL {X  -160.070, Y  +335.868, Z    +0.000, E1   +27.320, E3 +211924.236}
SPL {X  -163.969, Y  +354.959, Z    +0.000, E1   +17.178, E3 +211924.750}
SPL {X  -165.261, Y  +367.153, Z    +0.000, E1    +9.611, E3 +211923.903}
SPL {X  -165.600, Y  +374.440, Z    +0.000, E1    +4.699, E3 +211923.164}
SPL {X  -165.650, Y  +379.657, Z    +0.000, E1    +0.819, E3 +211922.693}
SPL {X  -165.650, Y  +381.885, Z    +0.000, E1    -1.282, E3 +211921.937}
SPL {X  -165.650, Y  +386.855, Z    +0.000, E1    -7.700, E3 +211921.356}
SPL {X  -165.650, Y  +393.198, Z    +0.000, E1   -17.733, E3 +211920.332}
SPL {X  -165.650, Y  +399.991, Z    +0.000, E1   -27.922, E3 +211921.227}
SPL {X  -165.650, Y  +409.148, Z    +0.000, E1   -43.235, E3 +211916.614}
SPL {X  -165.650, Y  +420.563, Z    +0.000, E1   -54.059, E3 +211917.172}
SPL {X  -165.650, Y  +436.566, Z    +0.000, E1   -62.888, E3 +211918.884}
SPL {X  -165.650, Y  +479.770, Z    +0.000, E1   -67.621, E3 +211938.223}
SPL {X  -165.650, Y  +594.725, Z    +0.000, E1   -69.155, E3 +212005.685}
ENDSPLINE

SPLINE
SPL {X  -165.650, Y  +565.175, Z    +0.000, E1   -62.653, E3 +212029.176}
ENDSPLINE

SPLINE
SPL {X  -165.650, Y  +576.067, Z    +0.000, E1   -62.373, E3 +212042.577}
SPL {X  -165.650, Y  +586.101, Z    +0.000, E1   -62.398, E3 +212053.159}
SPL {X  -165.650, Y  +596.110, Z    +0.000, E1   -62.302, E3 +212064.600}
SPL {X  -165.650, Y  +607.052, Z    +0.000, E1   -62.387, E3 +212075.667}
SPL {X  -165.650, Y  +618.920, Z    +0.000, E1   -62.340, E3 +212088.858}
SPL {X  -165.650, Y  +631.247, Z    +0.000, E1   -62.270, E3 +212102.474}
SPL {X  -165.650, Y  +645.288, Z    +0.000, E1   -62.475, E3 +212116.154}
SPL {X  -165.650, Y  +657.265, Z    +0.000, E1   -62.410, E3 +212129.273}
SPL {X  -165.650, Y  +665.926, Z    +0.000, E1   -62.171, E3 +212140.286}
SPL {X  -165.644, Y  +676.899, Z    +0.000, E1   -62.447, E3 +212150.054}
SPL {X  -165.241, Y  +687.133, Z    +0.000, E1   -62.230, E3 +212162.756}
SPL {X  -164.056, Y  +698.425, Z    +0.000, E1   -62.113, E3 +212175.573}
SPL {X  -162.891, Y  +705.608, Z    +0.000, E1   -61.899, E3 +212184.745}
SPL {X  -160.709, Y  +715.657, Z    +0.000, E1   -61.639, E3 +212197.496}
SPL {X  -157.706, Y  +726.183, Z    +0.000, E1   -61.153, E3 +212211.879}
SPL {X  -155.057, Y  +733.785, Z    +0.000, E1   -60.834, E3 +212221.869}
SPL {X  -152.882, Y  +739.274, Z    +0.000, E1   -60.485, E3 +212229.862}
SPL {X  -150.387, Y  +744.953, Z    +0.000, E1   -60.023, E3 +212238.537}
SPL {X  -146.839, Y  +752.170, Z    +0.000, E1   -59.458, E3 +212249.495}
SPL {X  -142.415, Y  +760.104, Z    +0.000, E1   -58.730, E3 +212261.554}
SPL {X  -132.386, Y  +775.068, Z    +0.000, E1   -61.559, E3 +212263.623}
SPL {X   -89.692, Y  +814.767, Z    +0.000, E1   -54.641, E3 +212377.672}
ENDSPLINE

